// SIMATIC STEP 7 (V5.x) project 450_DMC60U
// CPU: PLC317-2DP
// station: P_ADR_BUS
// station: Hardware
// station: SINUMERIK
// station: P_ADR_BUS
// station: Hardware
// station: KSM
// station: P_ADR_BUS
// station: Hardware
// station: Rüstplatztüre
// station: P_ADR_BUS
// station: Hardware
// station: Rüstplatz_AG
// program: S7-Programm(1)
// program: S7-Programm(1)
// program: S7-Programm(1)
// program: S7-Programm(8)
// program: SINUMERIK_NX15
// program: SINAMICS_In_NCU_720

SYMBOL_TABLE
"DB_MESSAGE"	DB 2	UDT 2	// Arbeitsdaten Alarm-/Meldungserfassung
"INST_DB_TOOLING_SYSTEM"	DB 15	FB 15	// Nullpunktspannsystem
"DB_COOLANT"	DB 50	UDT 50	// Kühlmittelanlage
"INS_MESSAGE_OUT"	DB 100	FB 100	// Arbeitsdaten Alarm-/Meldungserfassung
"DB_CK_OP"	DB 101	UDT 101	// DB für Überwachung von Operanden
"DB_IN"	DB 111	DB 111	// Kommunikation - Eingänge
"DB_OUT"	DB 112	DB 112	// Kommunikation - Ausgänge
"TOOLING SYSTEM???"	FB 15	FB 15	// Nullpunktspannsystem
"MESSAGE_OUT"	FB 100	FB 100	// Ausgabe Alarm-/Betriebsmeldungen
"FLOW_CONTROL"	FC 10	FC 10	// Durchflussüberwachung
"STATUS_INDICATOR"	FC 30	FC 30
"COOLANT"	FC 50	FC 50	// Kühlmittel Druckerhöhung
"FUNCTIONS"	FC 90	FC 90	// allgemeine Funktionen
"CHANGE_BYTE"	FC 91	FC 91
"SIGNAL"	FC 92	FC 92	// allgemeine Signalverknüpfungen
"FC_CK2OP"	FC 101	FC 101	// Überwachung von 2 Operanden
"FC_CK1OP"	FC 102	FC 102	// Überwachung eines Operanden
"INPUT_MASTER"	FC 111	FC 111	// Eingänge von Mastersystem lesen
"OUTPUT_MASTER"	FC 112	FC 112	// Ausgänge an Mastersystem schreiben
"INPUT_PERIPHERIE"	FC 121	FC 121	// Eingänge von Peripherie lesen
"OUTPUT_PERIPHERIE"	FC 122	FC 122	// Ausgänge an Peripherie schreiben
"M_LOW"	M 0.0	BOOL	// Merker mit Zustand Low  "FALSE"
"M_HIGH"	M 0.1	BOOL	// Merker mit Zustand High  "TRUE"
"m_expertenbit"	M 0.2	BOOL	// Expertenbit für Fehleranzeige
"M_STARTPULSE"	M 0.5	BOOL	// Startimpuls, wird nur einmalig, für einen Zyklus gesetzt.
"m_inbetriebnahme"	M 0.6	BOOL
"m_konstruktion"	M 0.7	BOOL
"M_TAKT_0.1SEC"	M 1.0	BOOL	// Taktmerker 0.1sec/10Hz
"M_TAKT_0.2SEC"	M 1.1	BOOL	// Taktmerker 0.2sec/5Hz
"M_TAKT_0.4SEC"	M 1.2	BOOL	// Taktmerker 0.4sec/2.5Hz
"M_TAKT_0.5SEC"	M 1.3	BOOL	// Taktmerker 0.5sec/2Hz
"M_TAKT_0.8SEC"	M 1.4	BOOL	// Taktmerker 0.8sec/1.25Hz
"M_TAKT_1.0SEC"	M 1.5	BOOL	// Taktmerker 1.0sec/1Hz
"M_TAKT_1.6SEC"	M 1.6	BOOL	// Taktmerker 1.6sec/0.625Hz
"M_TAKT_2.0SEC"	M 1.7	BOOL	// Taktmerker 2.0sec/0.5Hz
"Hilfsmerker_Flanke_1"	M 10.0	BOOL
"Hilfsmerker_Flanke_2"	M 10.1	BOOL
"Hilfsmerker_Flanke_3"	M 10.3	BOOL
"Hilfsmerker_Flanke_4"	M 10.4	BOOL
"Hilfsmerker_Flanke_5"	M 10.5	BOOL
"Hilfsmerker_Flanke_6"	M 10.6	BOOL
"Hilfsmerker_KSS_aus"	M 10.7	BOOL
"Hilfsmerker_KSS_aus1"	M 11.0	BOOL
"m_sqz"	M 11.1	BOOL	// zus.Störung quittieren
"m_ilp_ventilate"	M 11.2	BOOL	// Anlage belüftet
"m_need_ventilate"	M 11.3	BOOL	// Benötigt Entlüftung
"kmsto"	M 50.0	BOOL	// Kühlmittelanlage Sammelstörung
"m_fn_m7S"	M 50.1	BOOL	// negative Flanke von M7/Spritzpistole
"m_fp_masch_on"	M 50.2	BOOL	// positive Flanke bei Maschine Ein
"m_fn_m7opendoor"	M 50.3	BOOL	// negative Flanke von M7 bei öffnen der Arbeitsraumtüre
"m50.4"	M 50.4	BOOL
"m50.5"	M 50.5	BOOL
"m50.6"	M 50.6	BOOL
"m50.7"	M 50.7	BOOL
"m51.0"	M 51.0	BOOL
"m51.1"	M 51.1	BOOL
"m51.2"	M 51.2	BOOL
"m51.3"	M 51.3	BOOL
"m51.4"	M 51.4	BOOL
"m51.5"	M 51.5	BOOL
"m51.6"	M 51.6	BOOL
"m51.7"	M 51.7	BOOL
"m52.0"	M 52.0	BOOL
"m52.1"	M 52.1	BOOL
"m52.2"	M 52.2	BOOL
"m52.3"	M 52.3	BOOL
"m52.4"	M 52.4	BOOL
"m52.5"	M 52.5	BOOL
"m52.6"	M 52.6	BOOL
"m52.7"	M 52.7	BOOL
"m53.0"	M 53.0	BOOL
"m53.1"	M 53.1	BOOL
"m53.2"	M 53.2	BOOL
"m53.3"	M 53.3	BOOL
"m53.4"	M 53.4	BOOL
"m53.5"	M 53.5	BOOL
"m53.6"	M 53.6	BOOL
"m53.7"	M 53.7	BOOL
"m54.0"	M 54.0	BOOL
"m54.1"	M 54.1	BOOL
"m54.2"	M 54.2	BOOL
"m54.3"	M 54.3	BOOL
"m54.4"	M 54.4	BOOL
"m54.5"	M 54.5	BOOL
"m54.6"	M 54.6	BOOL
"m54.7"	M 54.7	BOOL
"m55.0"	M 55.0	BOOL
"m55.1"	M 55.1	BOOL
"m55.2"	M 55.2	BOOL
"m55.3"	M 55.3	BOOL
"m55.4"	M 55.4	BOOL
"m55.5"	M 55.5	BOOL
"m55.6"	M 55.6	BOOL
"m55.7"	M 55.7	BOOL
"m56.0"	M 56.0	BOOL
"m56.1"	M 56.1	BOOL
"m56.2"	M 56.2	BOOL
"m56.3"	M 56.3	BOOL
"m56.4"	M 56.4	BOOL
"m56.5"	M 56.5	BOOL
"m56.6"	M 56.6	BOOL
"m56.7"	M 56.7	BOOL
"m57.0"	M 57.0	BOOL
"m57.1"	M 57.1	BOOL
"m57.2"	M 57.2	BOOL
"m57.3"	M 57.3	BOOL
"m57.4"	M 57.4	BOOL
"m57.5"	M 57.5	BOOL
"m57.6"	M 57.6	BOOL
"m57.7"	M 57.7	BOOL
"m_pumpe_testlauf"	M 60.0	BOOL	// Start Niederdruckpumpe (für Testlauf)
"EPX_FLOW_HD"	M 100.0	BOOL	// Durchflusswächter Kühlmittel2 (M7)
"EPX_WIREBREAK_HD"	M 100.1	BOOL	// /Durchflusswächter HD Leitungsüberwachung
"EPX_FLOW_ND"	M 100.2	BOOL	// Durchflusswächter Kühlmittel1 (M8)
"EPX_WIREBREAK_ND"	M 100.3	BOOL	// /Durchflusswächter ND Leitungsüberwachung
"EPX_ZPS_RELEASE"	M 100.4	BOOL	// Nullpunktspannsystem lösen
"EPX_ZPS_LOCK"	M 100.5	BOOL	// Nullpunktspannsystem gesperrt
"EPX_ZPS_PRESSURE_MIN1"	M 100.6	BOOL	// Nullpunktspannsystem Drucküberwachung_1 Minimaldruck (p~0) = gespannt
"EPX_ZPS_PRESSURE_MIN2"	M 100.7	BOOL	// Nullpunktspannsystem Drucküberwachung_2 Minimaldruck (p~0) = gespannt
"EPX_ZPS_PRESSURE_MAX1"	M 101.0	BOOL	// Nullpunktspannsystem Drucküberwachung_1 Maximaldruck (p=max) = gelöst
"EPX_ZPS_PRESSURE_MAX2"	M 101.1	BOOL	// Nullpunktspannsystem Drucküberwachung_2 Maximaldruck (p=max) = gelöst
"EPX_COOLANT_LIMIT_VALUE"	M 101.2	BOOL	// /Füllstandsüberwachung im Sammelbehälter
"EPX_LUBRICATION_LEVEL"	M 101.3	BOOL	// Füllstandsüberwachung Schmierstoffaggregat
"EPX_ZPS_MODE_AUTO"	M 101.4	BOOL	// Nullpunktspannsystem in Betriebsart Automatik = Ansteuerung durch ext. Einheit
"EPX_ZPS_INTERLOCK_MIN1"	M 101.5	BOOL	// Nullpunktspannsystem - Verriegelungskontrolle Druck ~0 (drucklos)
"EPX_ZPS_INTERLOCK_MAX1"	M 101.6	BOOL	// Nullpunktspannsystem - Verriegelungskontrolle Druck vorhanden (=verriegelt)
"EPX_ZPS_DISTANCE_P_MIN1"	M 101.7	BOOL	// Nullpunktspannsystem - Auflagenkontrolle Druck ~0 (drucklos)
"EPX_ZPS_DISTANCE_P_MAX1"	M 102.0	BOOL	// Nullpunktspannsystem - Auflagenkontrolle Druck erreicht (Präzision vorhanden)
"EPX_ALARM_QUIT"	M 102.1	BOOL	// Rücksetzen der Fehlermeldung (z.B. Akustik)
"EPX_EL-CABINETDOOR1_OPEN"	M 102.2	BOOL	// Schaltschranktür(-kombination)_1 der Werkzeugmaschine geöffnet
"EPX_EL-CABINETDOOR2_OPEN"	M 102.3	BOOL	// Schaltschranktür(-kombination)_2 der Werkzeugmaschine geöffnet
"EPX_EL-CABINETDOOR5_OPEN"	M 102.4	BOOL	// Schaltschranktür(-kombination)_1 der Kühlschmierstoffanlage geöffnet
"EPX_EL_CABINET_TEMP_1"	M 102.5	BOOL	// Uebertemperatur Schaltschrank Werkzeugmaschine
"EPX_EL_CABINET_TEMP_2"	M 102.6	BOOL	// Grenzwertmeldung Schaltschranktemperatur Werkzeugmaschine
"EPX_EL-CABINETDOOR3_OPEN"	M 102.7	BOOL	// Schaltschranktür(-kombination)_3 der Werkzeugmaschine geöffnet
"EPX_SO_APC_POS_180"	M 103.0	BOOL	// Palettenwechsler Stellung 180 Grad (Palette_2 im Arbeitsraum)
"EPX_SO_APC_POS_0"	M 103.1	BOOL	// Palettenwechsler Stellung 0 Grad (Palette_1 im Arbeitsraum)
"EPX_VCS_MODE_MIXED"	M 103.2	BOOL	// Anwahl Betriebsart <Vakuumsystem Mischbetrieb> aktiv
"EPX_VCS_MODE_VACUUM"	M 103.3	BOOL	// Anwahl Betriebsart <Vakuumsystem Vollwechsel> aktiv
"EPX_VCS_MODE_OFF"	M 103.4	BOOL	// Anwahl Betriebsart <Vakuumsystem Aus>
"EPX_VCS_READY_1"	M 103.5	BOOL	// Betriebsbereitmeldung Vakuumsystem (Arbeitsraum) z.B. Leistungssschalter, ...
"EPX_VCS_READY_2"	M 103.6	BOOL	// Betriebsbereitmeldung Vakuumsystem (Rüstplatz) z.B. Leistungssschalter, ...
"EPX_VCS_RELEASE_FIXTURE2"	M 103.7	BOOL	// Vakuumspannsystem am Rüstplatz lösen
"EPX_VCS_FIXTURE1_1_P=0"	M 104.0	BOOL	// Vakuumspannsystem im Arbeitsraum Drucklos (=gelöst)
"EPX_VCS_FIXTURE1_2_P=0"	M 104.1	BOOL	// Vakuumspannsystem im Arbeitsraum Drucklos (=gelöst)
"EPX_VCS_FIXTURE2_1_P=0"	M 104.2	BOOL	// Vakuumspannsystem am Rüstplatz Drucklos (=gelöst)
"EPX_VCS_FIXTURE1_1_P=MAX"	M 104.3	BOOL	// Vakuumspannsystem im Arbeitsraum gespannt (eingestellter Sollwert erreicht)
"EPX_VCS_FIXTURE2_1_P=MAX"	M 104.4	BOOL	// Vakuumspannsystem am Rüstplatz gespannt (eingestellter Sollwert erreicht)
"EPX_NEG_HYD_FILTERALARM1"	M 104.5	BOOL	// Filterverschmutzung Hydraulikfilter-Maschine (Alarm 100%)
"EPX_NEG_HYD_FILTERWARN1"	M 104.6	BOOL	// Filterverschmutzung Hydraulikfilter-Maschine (Warnung 75%)
"EPX_NEG_FUSE_AIRFILTER"	M 104.7	BOOL	// Auswertung Leistungsschalter des Nebelabscheiders/Absaugung
"EPX_POWER_AIRFILTER"	M 105.0	BOOL	// Überwachung Ansteuerung Nebelabscheider
"EPX_MACHINE_ON_K1"	M 105.1	BOOL	// "Maschine Ein"-Signal an Kühlschmierstoffanlage (kein Not-Aus)
"EPX_WORKROOM_CLOSED_K1"	M 105.2	BOOL	// "Arbeitsraumtüren geschlossen"-Signal an Kühlschmierstoffanlage
"EPX_NEG_COO_MESSAGE"	M 105.3	BOOL	// Warnmeldung von Kühlschmierstoffanlage
"EPX_NEG_COO_ALARM"	M 105.4	BOOL	// Störung, Alarm von Kühlschmierstoffanlage
"EPX_COO_ACK_COOLANT2.2"	M 105.5	BOOL	// Rückmeldung wenn Druckstufe_2 von Kühlmittel_2 erreicht wurde (YD-Anlauf)
"EPX_COO_MAINVALVE_CLOSED"	M 105.6	BOOL	// Kühlschmierstoffzufuhr Haupt-/Zentralventil geschlossen
"EPX_COO_PRESSURE_P=MAX"	M 105.7	BOOL	// Kühlschmierstoffzufuhr Drucküberwachung
"EPX_COO_MAIN_FLOW"	M 106.0	BOOL	// Kühlschmierstoffzufuhr Durchflussüberwachung
"EPX_COO_LIMITVALUE_K5"	M 106.1	BOOL	// Grenzwertmeldung aus Sammelbehälter (SPF) z.B. von WHG-Sonde
"EPX_NEG_COO_FILTALARM2.2"	M 106.2	BOOL	// Filterverschmutzung Feinfilter Alarmmeldung für KSS-Zufuhr_2 (IKZ)-Druckstufe_2
"EPX_COO_FILTWARN2.2"	M 106.3	BOOL	// Filterverschmutzung Feinfilter Warnmeldung für KSS-Zufuhr_2 (IKZ) - Druckstufe_2
"EPX_VCS_RELEASE_FIXTURE1"	M 106.4	BOOL	// Vakuumspannsystem im Arbeitsraum lösen
"m106.5"	M 106.5	BOOL
"m106.6"	M 106.6	BOOL
"m106.7"	M 106.7	BOOL
"APX_SIGNAL_TOWER_GN"	M 180.0	BOOL	// Signalleuchte (Ampel) Element: GRÜN (GN)
"APX_SIGNAL_TOWER_YE"	M 180.1	BOOL	// Signalleuchte (Ampel) Element: GELB (YE)
"APX_SIGNAL_TOWER_RD"	M 180.2	BOOL	// Signalleuchte (Ampel) Element: ROT (RD)
"APX_BDE_AXIS_SPINDLE"	M 180.3	BOOL	// mindestens 1Achse und Spindel aktiv
"APX_BDE_MACHINE_ON"	M 180.4	BOOL	// Maschine Ein (kein Not-Aus)
"APX_MODE_MANUAL"	M 180.5	BOOL	// Betriebsart "MANUAL"
"APX_MODE_TEACH_IN"	M 180.6	BOOL	// Betriebsart "TEACH IN"
"APX_MODE_AUTOMATIK"	M 180.7	BOOL	// Betriebsart "AUTOMATIK"
"APX_FEEDRATE>X%"	M 181.0	BOOL	// Vorschubpotentiometer größer Wert "X"
"APX_CNC_ERROR"	M 181.1	BOOL	// Fehlermeldung CNC
"APX_PROG_STOP"	M 181.2	BOOL	// Programm Halt
"APX_PROG_RUN"	M 181.3	BOOL	// Programm läuft
"APX_CNC_READY2RUN"	M 181.4	BOOL	// CNC-Betriebsbereit
"APX_ZPS_BLOW_OUT"	M 181.5	BOOL	// Nullpunktspannsystem Blasluft (Reinigung)
"APX_ZPS_STATUS"	M 181.6	BOOL	// Nullpunktspannsystem Statusmeldung Betriebsartenanzeige
"APX_ZPS_RELEASE1"	M 181.7	BOOL	// Nullpunktspannsystem lösen (Ventil_1)
"APX_ZPS_RELEASE2"	M 182.0	BOOL	// Nullpunktspannsystem lösen (Ventil_2)
"APX_ZPS_INTERLOCK1"	M 182.4	BOOL	// Nullpunktspannsystem - Ansteuerung (Ventil) für Verriegelungskontrolle
"APX_ZPS_DISTANCE_CHECK1"	M 182.5	BOOL	// Nullpunktspannsystem - Ansteuerung (Ventil) für Auflagenkontrolle
"APX_WORKPIECE_COUNT"	M 182.6	BOOL	// Werkstück Zählimpuls
"APX_PRODUCTION"	M 182.7	BOOL	// Produktionssignal der Werkzeugmaschine/Maschine Produziert (Programm läuft)
"APX_PALLET-NR_BIT0"	M 183.0	BOOL	// Nummer der Palette Arbeitsraum 2^0 (=1)
"APX_PALLET-NR_BIT1"	M 183.1	BOOL	// Nummer der Palette Arbeitsraum 2^1 (=2)
"APX_PALLET-NR_BIT2"	M 183.2	BOOL	// Nummer der Palette Arbeitsraum 2^2 (=4)
"APX_PALLET-NR_BIT3"	M 183.3	BOOL	// Nummer der Palette Arbeitsraum 2^3 (=8)
"APX_ALARM_LIGHT"	M 183.4	BOOL	// Optische Anzeige einer Fehlermeldung
"APX_AUDIBLE_ALARM"	M 183.5	BOOL	// Akustische Ausgabe einer Fehlermeldung
"APX_VCS_RELEASE_FIXTURE1"	M 183.6	BOOL	// Vakuumspannsystem im Arbeitsraum Lösen (=drucklos)
"APX_VCS_RELEASE_FIXTURE2"	M 183.7	BOOL	// Vakuumspannsystem am Rüstplatz Lösen (=drucklos)
"APX_AIRFILTER_ON"	M 184.0	BOOL	// Aktivieren und evtl.verzögertes Abschalten des Nebelabscheiders
"APX_COO_COOLANT1_(M8)"	M 184.1	BOOL	// Aktivierung Kühlschmierstoffzufuhr_1 (externe - Spritzdüsen)
"APX_COO_PALLET_CARRIER"	M 184.2	BOOL	// Aktivierung Spänespülung Palettenträger (Umschaltung IKZ)
"APX_COO_WORKPIECE_1"	M 184.3	BOOL	// Aktivierung Spänespülung Werkstückreinigung (Dachspülung)
"APX_COO_SPRAYGUN"	M 184.4	BOOL	// Aktivierung Spritzpistole, Spülpistole
"APX_COO_WORKROOMDOOR"	M 184.5	BOOL	// Aktivierung Spänespülung Kabinentüre, Arbeitsraumtüre
"APX_COO_COOLANT2.2"	M 184.6	BOOL	// Aktivierung Kühlschmierstoffzufuhr_2 (IKZ) - Druckstufe_2
"APX_COO_MAINVALVE"	M 184.7	BOOL	// Aktivierung Kühlschmierstoffzufuhr Haupt-/Zentralventil
"APX_COO_LOCKVALVE_RET"	M 185.0	BOOL	// Aktivierung Sperrventil für Kühlschmierstoffrückführung aus Sammelbehälter (SPF)
"APX_ALARM_RESET"	M 185.1	BOOL	// Bei Betätigung der "Alarm-Quit-Taste (F10)" wird Ausgang gesetzt
"APX_NO_MACHINING"	M 185.2	BOOL	// MDE/BDE: keine Bearbeitung
"APX_INTO_PRODUCTION"	M 185.3	BOOL	// MDE/BDE: Produktionssignal
"APX_PROG_END"	M 185.4	BOOL	// Programm Ende
"m185.5"	M 185.5	BOOL
"m185.6"	M 185.6	BOOL
"m185.7"	M 185.7	BOOL
"APX_COO_LOCKVALVE2.2"	M 188.0	BOOL	// Aktivierung Sperrventil für Kühlschmierstoffzufuhr - Druckstufe_2
"QpxFlushSetUpStation"	M 197.0	BOOL	// Spänespülung am Rüstplatz (Spannvorrichtung, Werkstück, ...)
"m_AkTime"	MD 12	TIME	// ausgeleseneSysZeitVonTime_tck SFC64
"APW_COO_PRESS_VALUE2.2"	MW 186	WORD	// Sollwertvorgabe für Druckvorwahl Kühlmittel_2 (inner Kühlschmierstoffzufuhr)
"CYCL_EXC"	OB 1	OB 1	// Cycle Execution
"I/O_FLT1"	OB 82	OB 82	// I/O Point Fault 1
"CPU_FLT"	OB 84	OB 84	// CPU Fault
"OBNL_FLT"	OB 85	OB 85	// OB Not Loaded Fault
"RACK_FLT"	OB 86	OB 86	// Loss of Rack Fault
"START"	OB 100	OB 100	// Anlauf OB
"PROG_ERR"	OB 121	OB 121	// Programming Error
"MOD_ERR"	OB 122	OB 122	// Module Access Error
"BLKMOV"	SFC 20	SFC 20	// Copy Variables
"TIME_TCK"	SFC 64	SFC 64	// Time tics of period 10 ms
"t0"	T 0	TIMER	// 840D Grundprg.
"t1"	T 1	TIMER	// 840D Grundprg.
"t2"	T 2	TIMER	// 840D Grundprg.
"t3"	T 3	TIMER	// 840D Grundprg.
"t4"	T 4	TIMER	// 840D Grundprg.
"t5"	T 5	TIMER	// 840D Grundprg.
"t6"	T 6	TIMER	// 840D Grundprg.
"t7"	T 7	TIMER	// 840D Grundprg.
"t8"	T 8	TIMER	// 840D Grundprg.
"t9"	T 9	TIMER	// 840D Grundprg.
"t10"	T 10	TIMER
"Hilfs_Timer_1"	T 11	TIMER
"Hilfs_Timer_2"	T 12	TIMER
"Hilfs_Timer_3"	T 13	TIMER
"Hilfs_Timer_4"	T 14	TIMER
"Hilfs_Timer_5"	T 15	TIMER
"Hilfs_Timer_6"	T 16	TIMER
"t_sp_twa"	T 17	TIMER	// se Nullspannsystem Schrittkette Wartezeit
"t_sp_tue"	T 18	TIMER	// se Nullspannsystem Schrittkette Überwachungszeit (Reserve)
"t_nspgs"	T 19	TIMER	// se Nullspannsystem gespannt
"t_nspgsa"	T 20	TIMER	// sa Nullspannsystem gespannt
"t_nspgl"	T 21	TIMER	// se Nullspannsystem gelöst
"t_nspgla"	T 22	TIMER	// sa Nullspannsystem gelöst
"t23"	T 23	TIMER
"t24"	T 24	TIMER
"t_toggle"	T 25	TIMER	// Zeit für FB100 Anzeigeintervall
"t26"	T 26	TIMER
"t27"	T 27	TIMER
"t28"	T 28	TIMER
"t29"	T 29	TIMER
"t30"	T 30	TIMER
"t31"	T 31	TIMER
"ta_pressureless"	T 32	TIMER	// Belüften der Druckerhöhungsstation nach M7
"t33"	T 33	TIMER
"t34"	T 34	TIMER
"t35"	T 35	TIMER
"t36"	T 36	TIMER
"t37"	T 37	TIMER
"t38"	T 38	TIMER
"t39"	T 39	TIMER
"t40"	T 40	TIMER
"t41"	T 41	TIMER
"t42"	T 42	TIMER
"t43"	T 43	TIMER
"t44"	T 44	TIMER
"t45"	T 45	TIMER
"t46"	T 46	TIMER
"t47"	T 47	TIMER
"t48"	T 48	TIMER
"t49"	T 49	TIMER
"ta_kss_mainvalve"	T 50	TIMER	// Ausschaltverzögerung Km-Hauptventil ein
"t_kmfue"	T 51	TIMER	// se Überwachung Kühlmittelfilter
"t_kmFSp"	T 52	TIMER	// sa Km-Hochdruck-Sperrventil ein (=Frg.Hochdruck)
"t_kmrv"	T 53	TIMER	// se KmRückförderventil=Sperrventil öffnen
"ta_kss_km1"	T 54	TIMER	// Ausschaltverzögerung Kühlmittelanwahl (AKZ = M8)
"ta_kss_spraygun"	T 55	TIMER	// Ausschaltverzögerung für Spritzpistole
"ta_kss_workroomdoor"	T 56	TIMER	// Ausschaltverzögerung für Türspülung
"ta_kss_workpiece1"	T 57	TIMER	// Ausschaltverzögerung für Dachspülung (Werkstückspülung)
"te_aktiv_monit_pressure"	T 58	TIMER	// Einschaltverzögerung für Aktivierung Drucküberwachung
"ta_kss_setupstation"	T 59	TIMER	// Ausschaltverzögerung für Rüstplatzspülung(Vorrichtung)
"UDT_MESSAGE"	UDT 2	UDT 2	// UDT zu DB2 (Datenformat für Meldungen)
"UDT_COOLANT"	UDT 50	UDT 50	// UDT zu DB_COOLANT
"UDT101"	UDT 101	UDT 101
"UDT1010"	UDT 1010	UDT 1010	// UDT für UDT 101
"VAT_IN_dbw0"	VAT 1	
"VAT_IN_dbw2"	VAT 2	
"VAT_IN_dbw4"	VAT 3	
"VAT_IN_dbw6"	VAT 4	
"VAT_IN_dbw10_12"	VAT 5	
"VAT_OUT_dbw2"	VAT 6	
"VAT_OUT_dbw0"	VAT 7	
"VAT_PER"	VAT 8	
"VAT_MESSAGE"	VAT 9		// Meldungen, Alarme
"V_Nps0"	VAT 10		// Nullspannsystem
"V_allg"	VAT 11	
"VATksaÜW"	VAT 12	
"VAT_OUT_dbw6"	VAT 13	
END_SYMBOL_TABLE

TYPE "UDT_MESSAGE"	// UDT 2
AUTHOR : SPAC_slh
VERSION : 0.0
  STRUCT
   ALARM_001 : BOOL ;	//Schaltschranktemperatur zu hoch
   ALARM_002 : BOOL ;	//Schaltschranktemperatur - Grenzwert überschritten
   F003 : BOOL ;	//1-
   F004 : BOOL ;	//1-
   F005 : BOOL ;	//1-
   F006 : BOOL ;	//1-
   F007 : BOOL ;	//1-
   F008 : BOOL ;	//1-
   F009 : BOOL ;	//1-
   F010 : BOOL ;	//1-
   F011 : BOOL ;	//1-
   F012 : BOOL ;	//1-
   F013 : BOOL ;	//1-
   F014 : BOOL ;	//1-
   F015 : BOOL ;	//1-
   F016 : BOOL ;	//1-
   F017 : BOOL ;	//Nullpunktspannsysten Laufzeitfehler lösen_1
   F018 : BOOL ;	//Spanner 1 LzFehler spannen
   F019 : BOOL ;	//Spanner 1 Fehler Endlage gelöst
   F020 : BOOL ;	//Spanner 1 Fehler Endlage gespannt
   F021 : BOOL ;	//Spanner 1 Fehler Paarüberwachung
   F022 : BOOL ;	//Nullpunktspannsysten Laufzeitfehler lösen_2
   F023 : BOOL ;	//Spanner 2 LzFehler spannen
   F024 : BOOL ;	//Spanner 2 Fehler Endlage gelöst
   F025 : BOOL ;	//Spanner 2 Fehler Endlage gespannt
   F026 : BOOL ;	//Spanner 2 Fehler Paarüberwachung
   F027 : BOOL ;	//Auflagektrl.LzFehler bei einschalten
   F028 : BOOL ;	//Auflagektrl.LzFehler bei ausschalten
   F029 : BOOL ;	//Auflagektrl.Fehler Endlage Druck erreicht
   F030 : BOOL ;	//Auflagektrl.Fehler Endlage Drucklos
   F031 : BOOL ;	//Auflagektrl.Fehler Paarüberwachung
   F032 : BOOL ;	//Verriegelungsktrl.LzFehler bei einschalten
   F033 : BOOL ;	//Verriegelungsktrl.LzFehler bei ausschalten
   F034 : BOOL ;	//Verriegelungsktrl.Fehler Endlage Druck erreicht
   F035 : BOOL ;	//Verriegelungsktrl.Fehler Endlage Drucklos
   F036 : BOOL ;	//Verriegelungsktrl.Fehler Paarüberwachung
   F037 : BOOL ;	//1-
   F038 : BOOL ;	//1-
   F039 : BOOL ;	//1-
   F040 : BOOL ;	//1-
   F041 : BOOL ;	//1-
   F042 : BOOL ;	//1-
   F043 : BOOL ;	//1-
   F044 : BOOL ;	//1-
   F045 : BOOL ;	//1-
   F046 : BOOL ;	//1-
   F047 : BOOL ;	//1-
   F048 : BOOL ;	//1-
   F049 : BOOL ;	//1-
   F050 : BOOL ;	//1-
   F051 : BOOL ;	//1-
   F052 : BOOL ;	//1-
   F053 : BOOL ;	//1-
   F054 : BOOL ;	//1-
   F055 : BOOL ;	//1-
   F056 : BOOL ;	//1-
   F057 : BOOL ;	//1-
   F058 : BOOL ;	//1-
   F059 : BOOL ;	//1-
   F060 : BOOL ;	//1-
   F061 : BOOL ;	//1-
   F062 : BOOL ;	//1-
   F063 : BOOL ;	//1-
   F064 : BOOL ;	//1-
   F065 : BOOL ;	//1-
   F066 : BOOL ;	//1-
   F067 : BOOL ;	//1-
   F068 : BOOL ;	//1-
   F069 : BOOL ;	//1-
   F070 : BOOL ;	//1-
   F071 : BOOL ;	//1-
   F072 : BOOL ;	//1-
   F073 : BOOL ;	//1-
   F074 : BOOL ;	//1-
   F075 : BOOL ;	//1-
   F076 : BOOL ;	//1-
   F077 : BOOL ;	//1-
   F078 : BOOL ;	//1-
   F079 : BOOL ;	//1-
   F080 : BOOL ;	//1-
   F081 : BOOL ;	//1-
   F082 : BOOL ;	//1-
   F083 : BOOL ;	//1-
   F084 : BOOL ;	//1-
   F085 : BOOL ;	//1-
   F086 : BOOL ;	//1-
   F087 : BOOL ;	//1-
   F088 : BOOL ;	//1-
   F089 : BOOL ;	//1-
   F090 : BOOL ;	//1-
   F091 : BOOL ;	//1-
   F092 : BOOL ;	//1-
   F093 : BOOL ;	//1-
   F094 : BOOL ;	//1-
   F095 : BOOL ;	//1-
   F096 : BOOL ;	//1-
   F097 : BOOL ;	//Km-Hautpventil nicht offen, Eingang meldet "zu", muss 0-Signal melden
   F098 : BOOL ;	//Km-Hautpventil schließt nicht, Eingang muss 1-Signal melden
   F099 : BOOL ;	//WHG-Alarm
   F100 : BOOL ;	//Reserve Km-Alarm
   F101 : BOOL ;	//Km-Systemdruck fehlt, Eingang muss 1-Signal melden
   F102 : BOOL ;	//Km-Systemdruck, Druckschalter defekt, Eingang muss 0-Signal melden
   F103 : BOOL ;	//Km-Durchfluss fehlt, Eingang muss 1-Signal melden
   F104 : BOOL ;	//Km-Durchfluss-Schalter defekt, Eingang muss 0-Signal melden
   F105 : BOOL ;	//Kühlmittelfeinfilter verschmutzt
   F106 : BOOL ;	//Kühlmittelfeinfilter Schalterpaarüberwachung
   F107 : BOOL ;	//Reserve Km-Alarm
   F108 : BOOL ;	//Reserve Km-Alarm
   F109 : BOOL ;	//Reserve Km-Alarm
   F110 : BOOL ;	//Reserve Km-Alarm
   F111 : BOOL ;	//Reserve Km-Alarm
   F112 : BOOL ;	//Reserve Km-Alarm
   F113 : BOOL ;	//1-
   F114 : BOOL ;	//1-
   F115 : BOOL ;	//1-
   F116 : BOOL ;	//1-
   F117 : BOOL ;	//1-
   F118 : BOOL ;	//1-
   F119 : BOOL ;	//1-
   F120 : BOOL ;	//1-
   F121 : BOOL ;	//1-
   F122 : BOOL ;	//1-
   F123 : BOOL ;	//1-
   F124 : BOOL ;	//1-
   F125 : BOOL ;	//1-
   F126 : BOOL ;	//1-
   F127 : BOOL ;	//1-
   F128 : BOOL ;	//1-
   F129 : BOOL ;	//1-
   F130 : BOOL ;	//1-
   F131 : BOOL ;	//1-
   F132 : BOOL ;	//1-
   F133 : BOOL ;	//1-
   F134 : BOOL ;	//1-
   F135 : BOOL ;	//1-
   F136 : BOOL ;	//1-
   F137 : BOOL ;	//1-
   F138 : BOOL ;	//1-
   F139 : BOOL ;	//1-
   F140 : BOOL ;	//1-
   F141 : BOOL ;	//1-
   F142 : BOOL ;	//1-
   F143 : BOOL ;	//1-
   F144 : BOOL ;	//1-
   F145 : BOOL ;	//1-
   F146 : BOOL ;	//1-
   F147 : BOOL ;	//1-
   F148 : BOOL ;	//1-
   F149 : BOOL ;	//1-
   F150 : BOOL ;	//1-
   F151 : BOOL ;	//1-
   F152 : BOOL ;	//1-
   F153 : BOOL ;	//1-
   F154 : BOOL ;	//1-
   F155 : BOOL ;	//1-
   F156 : BOOL ;	//1-
   F157 : BOOL ;	//1-
   F158 : BOOL ;	//1-
   F159 : BOOL ;	//1-
   F160 : BOOL ;	//1-
   F161 : BOOL ;	//1-
   F162 : BOOL ;	//1-
   F163 : BOOL ;	//1-
   F164 : BOOL ;	//1-
   F165 : BOOL ;	//1-
   F166 : BOOL ;	//1-
   F167 : BOOL ;	//1-
   F168 : BOOL ;	//1-
   F169 : BOOL ;	//1-
   F170 : BOOL ;	//1-
   F171 : BOOL ;	//1-
   F172 : BOOL ;	//1-
   F173 : BOOL ;	//1-
   F174 : BOOL ;	//1-
   F175 : BOOL ;	//1-
   F176 : BOOL ;	//1-
   F177 : BOOL ;	//1-
   F178 : BOOL ;	//1-
   F179 : BOOL ;	//1-
   F180 : BOOL ;	//1-
   F181 : BOOL ;	//1-
   F182 : BOOL ;	//1-
   F183 : BOOL ;	//1-
   F184 : BOOL ;	//1-
   F185 : BOOL ;	//1-
   F186 : BOOL ;	//1-
   F187 : BOOL ;	//1-
   F188 : BOOL ;	//1-
   F189 : BOOL ;	//1-
   F190 : BOOL ;	//1-
   F191 : BOOL ;	//1-
   F192 : BOOL ;	//1-
   F193 : BOOL ;	//1-
   F194 : BOOL ;	//1-
   F195 : BOOL ;	//1-
   F196 : BOOL ;	//1-
   F197 : BOOL ;	//1-
   F198 : BOOL ;	//1-
   F199 : BOOL ;	//1-
   F200 : BOOL ;	//1-
   F201 : BOOL ;	//1-
   F202 : BOOL ;	//1-
   F203 : BOOL ;	//1-
   F204 : BOOL ;	//1-
   F205 : BOOL ;	//1-
   F206 : BOOL ;	//1-
   F207 : BOOL ;	//1-
   F208 : BOOL ;	//1-
   F209 : BOOL ;	//1-
   F210 : BOOL ;	//1-
   F211 : BOOL ;	//1-
   F212 : BOOL ;	//1-
   F213 : BOOL ;	//1-
   F214 : BOOL ;	//1-
   F215 : BOOL ;	//1-
   F216 : BOOL ;	//1-
   F217 : BOOL ;	//1-
   F218 : BOOL ;	//1-
   F219 : BOOL ;	//1-
   F220 : BOOL ;	//1-
   F221 : BOOL ;	//1-
   F222 : BOOL ;	//1-
   F223 : BOOL ;	//1-
   F224 : BOOL ;	//1-
   F225 : BOOL ;	//1-
   F226 : BOOL ;	//1-
   F227 : BOOL ;	//1-
   F228 : BOOL ;	//1-
   F229 : BOOL ;	//1-
   F230 : BOOL ;	//1-
   F231 : BOOL ;	//1-
   F232 : BOOL ;	//1-
   F233 : BOOL ;	//1-
   F234 : BOOL ;	//1-
   F235 : BOOL ;	//1-
   F236 : BOOL ;	//1-
   F237 : BOOL ;	//1-
   F238 : BOOL ;	//1-
   F239 : BOOL ;	//1-
   F240 : BOOL ;	//1-
   F241 : BOOL ;	//1-
   F242 : BOOL ;	//1-
   F243 : BOOL ;	//1-
   F244 : BOOL ;	//1-
   F245 : BOOL ;	//1-
   F246 : BOOL ;	//1-
   F247 : BOOL ;	//1-
   F248 : BOOL ;	//1-
   F249 : BOOL ;	//1-
   F250 : BOOL ;	//1-
   F251 : BOOL ;	//1-
   F252 : BOOL ;	//1-
   F253 : BOOL ;	//1-
   F254 : BOOL ;	//1-
   F255 : BOOL ;	//1-
   F256 : BOOL ;	//1-
   F257 : BOOL ;	//1-
   F258 : BOOL ;	//1-
   F259 : BOOL ;	//1-
   F260 : BOOL ;	//1-
   F261 : BOOL ;	//1-
   F262 : BOOL ;	//1-
   F263 : BOOL ;	//1-
   F264 : BOOL ;	//1-
   F265 : BOOL ;	//1-
   F266 : BOOL ;	//1-
   F267 : BOOL ;	//1-
   F268 : BOOL ;	//1-
   F269 : BOOL ;	//1-
   F270 : BOOL ;	//1-
   F271 : BOOL ;	//1-
   F272 : BOOL ;	//1-
   F273 : BOOL ;	//1-
   F274 : BOOL ;	//1-
   F275 : BOOL ;	//1-
   F276 : BOOL ;	//1-
   F277 : BOOL ;	//1-
   F278 : BOOL ;	//1-
   F279 : BOOL ;	//1-
   F280 : BOOL ;	//1-
   F281 : BOOL ;	//1-
   F282 : BOOL ;	//1-
   F283 : BOOL ;	//1-
   F284 : BOOL ;	//1-
   F285 : BOOL ;	//1-
   F286 : BOOL ;	//1-
   F287 : BOOL ;	//1-
   F288 : BOOL ;	//1-
   F289 : BOOL ;	//1-
   F290 : BOOL ;	//1-
   F291 : BOOL ;	//1-
   F292 : BOOL ;	//1-
   F293 : BOOL ;	//1-
   F294 : BOOL ;	//1-
   F295 : BOOL ;	//1-
   F296 : BOOL ;	//1-
   F297 : BOOL ;	//1-
   F298 : BOOL ;	//1-
   F299 : BOOL ;	//1-
   F300 : BOOL ;	//1-
   F301 : BOOL ;	//1-
   F302 : BOOL ;	//1-
   F303 : BOOL ;	//1-
   F304 : BOOL ;	//1-
   F305 : BOOL ;	//1-
   F306 : BOOL ;	//1-
   F307 : BOOL ;	//1-
   F308 : BOOL ;	//1-
   F309 : BOOL ;	//1-
   F310 : BOOL ;	//1-
   F311 : BOOL ;	//1-
   F312 : BOOL ;	//1-
   F313 : BOOL ;	//1-
   F314 : BOOL ;	//1-
   F315 : BOOL ;	//1-
   F316 : BOOL ;	//1-
   F317 : BOOL ;	//1-
   F318 : BOOL ;	//1-
   F319 : BOOL ;	//1-
   F320 : BOOL ;	//1-
   F321 : BOOL ;	//1-
   F322 : BOOL ;	//1-
   F323 : BOOL ;	//1-
   F324 : BOOL ;	//1-
   F325 : BOOL ;	//1-
   F326 : BOOL ;	//1-
   F327 : BOOL ;	//1-
   F328 : BOOL ;	//1-
   F329 : BOOL ;	//1-
   F330 : BOOL ;	//1-
   F331 : BOOL ;	//1-
   F332 : BOOL ;	//1-
   F333 : BOOL ;	//1-
   F334 : BOOL ;	//1-
   F335 : BOOL ;	//1-
   F336 : BOOL ;	//1-
   F337 : BOOL ;	//1-
   F338 : BOOL ;	//1-
   F339 : BOOL ;	//1-
   F340 : BOOL ;	//1-
   F341 : BOOL ;	//1-
   F342 : BOOL ;	//1-
   F343 : BOOL ;	//1-
   F344 : BOOL ;	//1-
   F345 : BOOL ;	//1-
   F346 : BOOL ;	//1-
   F347 : BOOL ;	//1-
   F348 : BOOL ;	//1-
   F349 : BOOL ;	//1-
   F350 : BOOL ;	//1-
   F351 : BOOL ;	//1-
   F352 : BOOL ;	//1-
   F353 : BOOL ;	//1-
   F354 : BOOL ;	//1-
   F355 : BOOL ;	//1-
   F356 : BOOL ;	//1-
   F357 : BOOL ;	//1-
   F358 : BOOL ;	//1-
   F359 : BOOL ;	//1-
   F360 : BOOL ;	//1-
   F361 : BOOL ;	//1-
   F362 : BOOL ;	//1-
   F363 : BOOL ;	//1-
   F364 : BOOL ;	//1-
   F365 : BOOL ;	//1-
   F366 : BOOL ;	//1-
   F367 : BOOL ;	//1-
   F368 : BOOL ;	//1-
   F369 : BOOL ;	//1-
   F370 : BOOL ;	//1-
   F371 : BOOL ;	//1-
   F372 : BOOL ;	//1-
   F373 : BOOL ;	//1-
   F374 : BOOL ;	//1-
   F375 : BOOL ;	//1-
   F376 : BOOL ;	//1-
   F377 : BOOL ;	//1-
   F378 : BOOL ;	//1-
   F379 : BOOL ;	//1-
   F380 : BOOL ;	//1-
   F381 : BOOL ;	//1-
   F382 : BOOL ;	//1-
   F383 : BOOL ;	//1-
   F384 : BOOL ;	//1-
   F385 : BOOL ;	//1-
   F386 : BOOL ;	//1-
   F387 : BOOL ;	//1-
   F388 : BOOL ;	//1-
   F389 : BOOL ;	//1-
   F390 : BOOL ;	//1-
   F391 : BOOL ;	//1-
   F392 : BOOL ;	//1-
   F393 : BOOL ;	//1-
   F394 : BOOL ;	//1-
   F395 : BOOL ;	//1-
   F396 : BOOL ;	//1-
   F397 : BOOL ;	//1-
   F398 : BOOL ;	//1-
   F399 : BOOL ;	//1-
   F400 : BOOL ;	//1-
   F401 : BOOL ;	//1-
   F402 : BOOL ;	//1-
   F403 : BOOL ;	//1-
   F404 : BOOL ;	//1-
   F405 : BOOL ;	//1-
   F406 : BOOL ;	//1-
   F407 : BOOL ;	//1-
   F408 : BOOL ;	//1-
   F409 : BOOL ;	//1-
   F410 : BOOL ;	//1-
   F411 : BOOL ;	//1-
   F412 : BOOL ;	//1-
   F413 : BOOL ;	//1-
   F414 : BOOL ;	//1-
   F415 : BOOL ;	//1-
   F416 : BOOL ;	//1-
   F417 : BOOL ;	//1-
   F418 : BOOL ;	//1-
   F419 : BOOL ;	//1-
   F420 : BOOL ;	//1-
   F421 : BOOL ;	//1-
   F422 : BOOL ;	//1-
   F423 : BOOL ;	//1-
   F424 : BOOL ;	//1-
   F425 : BOOL ;	//1-
   F426 : BOOL ;	//1-
   F427 : BOOL ;	//1-
   F428 : BOOL ;	//1-
   F429 : BOOL ;	//1-
   F430 : BOOL ;	//1-
   F431 : BOOL ;	//1-
   F432 : BOOL ;	//1-
   F433 : BOOL ;	//1-
   F434 : BOOL ;	//1-
   F435 : BOOL ;	//1-
   F436 : BOOL ;	//1-
   F437 : BOOL ;	//1-
   F438 : BOOL ;	//1-
   F439 : BOOL ;	//1-
   F440 : BOOL ;	//1-
   F441 : BOOL ;	//1-
   F442 : BOOL ;	//1-
   F443 : BOOL ;	//1-
   F444 : BOOL ;	//1-
   F445 : BOOL ;	//1-
   F446 : BOOL ;	//1-
   F447 : BOOL ;	//1-
   F448 : BOOL ;	//1-
   F449 : BOOL ;	//1-
   F450 : BOOL ;	//1-
   F451 : BOOL ;	//1-
   F452 : BOOL ;	//1-
   F453 : BOOL ;	//1-
   F454 : BOOL ;	//1-
   F455 : BOOL ;	//1-
   F456 : BOOL ;	//1-
   F457 : BOOL ;	//1-
   F458 : BOOL ;	//1-
   F459 : BOOL ;	//1-
   F460 : BOOL ;	//1-
   F461 : BOOL ;	//1-
   F462 : BOOL ;	//1-
   F463 : BOOL ;	//1-
   F464 : BOOL ;	//1-
   F465 : BOOL ;	//1-
   F466 : BOOL ;	//1-
   F467 : BOOL ;	//1-
   F468 : BOOL ;	//1-
   F469 : BOOL ;	//1-
   F470 : BOOL ;	//1-
   F471 : BOOL ;	//1-
   F472 : BOOL ;	//1-
   F473 : BOOL ;	//1-
   F474 : BOOL ;	//1-
   F475 : BOOL ;	//1-
   F476 : BOOL ;	//1-
   F477 : BOOL ;	//1-
   F478 : BOOL ;	//1-
   F479 : BOOL ;	//1-
   F480 : BOOL ;	//1-
   F481 : BOOL ;	//1-
   F482 : BOOL ;	//1-
   F483 : BOOL ;	//1-
   F484 : BOOL ;	//1-
   F485 : BOOL ;	//1-
   F486 : BOOL ;	//1-
   F487 : BOOL ;	//1-
   F488 : BOOL ;	//1-
   F489 : BOOL ;	//1-
   F490 : BOOL ;	//1-
   F491 : BOOL ;	//1-
   F492 : BOOL ;	//1-
   F493 : BOOL ;	//1-
   F494 : BOOL ;	//1-
   F495 : BOOL ;	//1-
   F496 : BOOL ;	//1-
   F497 : BOOL ;	//1-
   F498 : BOOL ;	//1-
   F499 : BOOL ;	//1-
   F500 : BOOL ;	//1-
   F501 : BOOL ;	//1-
   F502 : BOOL ;	//1-
   F503 : BOOL ;	//1-
   F504 : BOOL ;	//1-
   F505 : BOOL ;	//1-
   F506 : BOOL ;	//1-
   F507 : BOOL ;	//1-
   F508 : BOOL ;	//1-
   F509 : BOOL ;	//1-
   F510 : BOOL ;	//1-
   F511 : BOOL ;	//1-
   F512 : BOOL ;	//1-
   MSG_513 : BOOL ;	//Schaltschranktüre(n) an Werkzeugmaschine geöffnet
   MSG_514 : BOOL ;	//Schaltschranktüre(n) an Kühlschmierstoffanlage geöffnet
   MSG_515 : BOOL ;	//Schaltschranktemperatur zu hoch
   Me516 : BOOL ;	//1-
   Me517 : BOOL ;	//1-
   Me518 : BOOL ;	//1-
   Me519 : BOOL ;	//1-
   Me520 : BOOL ;	//1-
   Me521 : BOOL ;	//1-
   Me522 : BOOL ;	//1-
   Me523 : BOOL ;	//1-
   Me524 : BOOL ;	//1-
   Me525 : BOOL ;	//1-
   Me526 : BOOL ;	//1-
   Me527 : BOOL ;	//1-
   Me528 : BOOL ;	//1-
   Me529 : BOOL ;	//1-
   Me530 : BOOL ;	//1-
   Me531 : BOOL ;	//1-
   Me532 : BOOL ;	//1-
   Me533 : BOOL ;	//1-
   Me534 : BOOL ;	//1-
   Me535 : BOOL ;	//1-
   Me536 : BOOL ;	//1-
   Me537 : BOOL ;	//1-
   Me538 : BOOL ;	//1-
   Me539 : BOOL ;	//1-
   Me540 : BOOL ;	//1-
   Me541 : BOOL ;	//1-
   Me542 : BOOL ;	//1-
   Me543 : BOOL ;	//1-
   Me544 : BOOL ;	//1-
   Me545 : BOOL ;	//1-
   Me546 : BOOL ;	//1-
   Me547 : BOOL ;	//1-
   Me548 : BOOL ;	//1-
   Me549 : BOOL ;	//1-
   Me550 : BOOL ;	//1-
   Me551 : BOOL ;	//1-
   Me552 : BOOL ;	//1-
   Me553 : BOOL ;	//1-
   Me554 : BOOL ;	//1-
   Me555 : BOOL ;	//1-
   Me556 : BOOL ;	//1-
   Me557 : BOOL ;	//1-
   Me558 : BOOL ;	//1-
   Me559 : BOOL ;	//1-
   Me560 : BOOL ;	//1-
   MSG_561 : BOOL ;	//ext.Km-Anlage:Warnung steht an
   MSG_562 : BOOL ;	//Warnung:Kühlmittelfeinfilter verschmutzt E10.2
   MSG_563 : BOOL ;	//Druckvorgabe von LPlc nicht übernommen da nicht in Toleranz
   Me564 : BOOL ;	//1-
   Me565 : BOOL ;	//1-
   Me566 : BOOL ;	//1-
   Me567 : BOOL ;	//1-
   Me568 : BOOL ;	//1-
   Me569 : BOOL ;	//1-
   Me570 : BOOL ;	//1-
   Me571 : BOOL ;	//1-
   Me572 : BOOL ;	//1-
   Me573 : BOOL ;	//1-
   Me574 : BOOL ;	//1-
   Me575 : BOOL ;	//1-
   Me576 : BOOL ;	//1-
   Me577 : BOOL ;	//1-
   Me578 : BOOL ;	//1-
   Me579 : BOOL ;	//1-
   Me580 : BOOL ;	//1-
   Me581 : BOOL ;	//1-
   Me582 : BOOL ;	//1-
   Me583 : BOOL ;	//1-
   Me584 : BOOL ;	//1-
   Me585 : BOOL ;	//1-
   Me586 : BOOL ;	//1-
   Me587 : BOOL ;	//1-
   Me588 : BOOL ;	//1-
   Me589 : BOOL ;	//1-
   Me590 : BOOL ;	//1-
   Me591 : BOOL ;	//1-
   Me592 : BOOL ;	//1-
   Me593 : BOOL ;	//1-
   Me594 : BOOL ;	//1-
   Me595 : BOOL ;	//1-
   Me596 : BOOL ;	//1-
   Me597 : BOOL ;	//1-
   Me598 : BOOL ;	//1-
   Me599 : BOOL ;	//1-
   Me600 : BOOL ;	//1-
   Me601 : BOOL ;	//1-
   Me602 : BOOL ;	//1-
   Me603 : BOOL ;	//1-
   Me604 : BOOL ;	//1-
   Me605 : BOOL ;	//1-
   Me606 : BOOL ;	//1-
   Me607 : BOOL ;	//1-
   Me608 : BOOL ;	//1-
   Me609 : BOOL ;	//1-
   Me610 : BOOL ;	//1-
   Me611 : BOOL ;	//1-
   Me612 : BOOL ;	//1-
   Me613 : BOOL ;	//1-
   Me614 : BOOL ;	//1-
   Me615 : BOOL ;	//1-
   Me616 : BOOL ;	//1-
   Me617 : BOOL ;	//1-
   Me618 : BOOL ;	//1-
   Me619 : BOOL ;	//1-
   Me620 : BOOL ;	//1-
   Me621 : BOOL ;	//1-
   Me622 : BOOL ;	//1-
   Me623 : BOOL ;	//1-
   Me624 : BOOL ;	//1-
   Me625 : BOOL ;	//1-
   Me626 : BOOL ;	//1-
   Me627 : BOOL ;	//1-
   Me628 : BOOL ;	//1-
   Me629 : BOOL ;	//1-
   Me630 : BOOL ;	//1-
   Me631 : BOOL ;	//1-
   Me632 : BOOL ;	//1-
   Me633 : BOOL ;	//1-
   Me634 : BOOL ;	//1-
   Me635 : BOOL ;	//1-
   Me636 : BOOL ;	//1-
   Me637 : BOOL ;	//1-
   Me638 : BOOL ;	//1-
   Me639 : BOOL ;	//1-
   Me640 : BOOL ;	//1-
   Me641 : BOOL ;	//1-
   Me642 : BOOL ;	//1-
   Me643 : BOOL ;	//1-
   Me644 : BOOL ;	//1-
   Me645 : BOOL ;	//1-
   Me646 : BOOL ;	//1-
   Me647 : BOOL ;	//1-
   Me648 : BOOL ;	//1-
   Me649 : BOOL ;	//1-
   Me650 : BOOL ;	//1-
   Me651 : BOOL ;	//1-
   Me652 : BOOL ;	//1-
   Me653 : BOOL ;	//1-
   Me654 : BOOL ;	//1-
   Me655 : BOOL ;	//1-
   Me656 : BOOL ;	//1-
   Me657 : BOOL ;	//1-
   Me658 : BOOL ;	//1-
   Me659 : BOOL ;	//1-
   Me660 : BOOL ;	//1-
   Me661 : BOOL ;	//1-
   Me662 : BOOL ;	//1-
   Me663 : BOOL ;	//1-
   Me664 : BOOL ;	//1-
   Me665 : BOOL ;	//1-
   Me666 : BOOL ;	//1-
   Me667 : BOOL ;	//1-
   Me668 : BOOL ;	//1-
   Me669 : BOOL ;	//1-
   Me670 : BOOL ;	//1-
   Me671 : BOOL ;	//1-
   Me672 : BOOL ;	//1-
   Me673 : BOOL ;	//1-
   Me674 : BOOL ;	//1-
   Me675 : BOOL ;	//1-
   Me676 : BOOL ;	//1-
   Me677 : BOOL ;	//1-
   Me678 : BOOL ;	//1-
   Me679 : BOOL ;	//1-
   Me680 : BOOL ;	//1-
   Me681 : BOOL ;	//1-
   Me682 : BOOL ;	//1-
   Me683 : BOOL ;	//1-
   Me684 : BOOL ;	//1-
   Me685 : BOOL ;	//1-
   Me686 : BOOL ;	//1-
   Me687 : BOOL ;	//1-
   Me688 : BOOL ;	//1-
   Me689 : BOOL ;	//1-
   Me690 : BOOL ;	//1-
   Me691 : BOOL ;	//1-
   Me692 : BOOL ;	//1-
   Me693 : BOOL ;	//1-
   Me694 : BOOL ;	//1-
   Me695 : BOOL ;	//1-
   Me696 : BOOL ;	//1-
   Me697 : BOOL ;	//1-
   Me698 : BOOL ;	//1-
   Me699 : BOOL ;	//1-
   Me700 : BOOL ;	//1-
   Me701 : BOOL ;	//1-
   Me702 : BOOL ;	//1-
   Me703 : BOOL ;	//1-
   Me704 : BOOL ;	//1-
   Me705 : BOOL ;	//1-
   Me706 : BOOL ;	//1-
   Me707 : BOOL ;	//1-
   Me708 : BOOL ;	//1-
   Me709 : BOOL ;	//1-
   Me710 : BOOL ;	//1-
   Me711 : BOOL ;	//1-
   Me712 : BOOL ;	//1-
   Me713 : BOOL ;	//1-
   Me714 : BOOL ;	//1-
   Me715 : BOOL ;	//1-
   Me716 : BOOL ;	//1-
   Me717 : BOOL ;	//1-
   Me718 : BOOL ;	//1-
   Me719 : BOOL ;	//1-
   Me720 : BOOL ;	//1-
   Me721 : BOOL ;	//1-
   Me722 : BOOL ;	//1-
   Me723 : BOOL ;	//1-
   Me724 : BOOL ;	//1-
   Me725 : BOOL ;	//1-
   Me726 : BOOL ;	//1-
   Me727 : BOOL ;	//1-
   Me728 : BOOL ;	//1-
   Me729 : BOOL ;	//1-
   Me730 : BOOL ;	//1-
   Me731 : BOOL ;	//1-
   Me732 : BOOL ;	//1-
   Me733 : BOOL ;	//1-
   Me734 : BOOL ;	//1-
   Me735 : BOOL ;	//1-
   Me736 : BOOL ;	//1-
   Me737 : BOOL ;	//1-
   Me738 : BOOL ;	//1-
   Me739 : BOOL ;	//1-
   Me740 : BOOL ;	//1-
   Me741 : BOOL ;	//1-
   Me742 : BOOL ;	//1-
   Me743 : BOOL ;	//1-
   Me744 : BOOL ;	//1-
   Me745 : BOOL ;	//1-
   Me746 : BOOL ;	//1-
   Me747 : BOOL ;	//1-
   Me748 : BOOL ;	//1-
   Me749 : BOOL ;	//1-
   Me750 : BOOL ;	//1-
   Me751 : BOOL ;	//1-
   Me752 : BOOL ;	//1-
   Me753 : BOOL ;	//1-
   Me754 : BOOL ;	//1-
   Me755 : BOOL ;	//1-
   Me756 : BOOL ;	//1-
   Me757 : BOOL ;	//1-
   Me758 : BOOL ;	//1-
   Me759 : BOOL ;	//1-
   Me760 : BOOL ;	//1-
   Me761 : BOOL ;	//1-
   Me762 : BOOL ;	//1-
   Me763 : BOOL ;	//1-
   Me764 : BOOL ;	//1-
   Me765 : BOOL ;	//1-
   Me766 : BOOL ;	//1-
   Me767 : BOOL ;	//1-
   Me768 : BOOL ;	//1-
   Me769 : BOOL ;	//1-
   Me770 : BOOL ;	//1-
   Me771 : BOOL ;	//1-
   Me772 : BOOL ;	//1-
   Me773 : BOOL ;	//1-
   Me774 : BOOL ;	//1-
   Me775 : BOOL ;	//1-
   Me776 : BOOL ;	//1-
   Me777 : BOOL ;	//1-
   Me778 : BOOL ;	//1-
   Me779 : BOOL ;	//1-
   Me780 : BOOL ;	//1-
   Me781 : BOOL ;	//1-
   Me782 : BOOL ;	//1-
   Me783 : BOOL ;	//1-
   Me784 : BOOL ;	//1-
   Me785 : BOOL ;	//1-
   Me786 : BOOL ;	//1-
   Me787 : BOOL ;	//1-
   Me788 : BOOL ;	//1-
   Me789 : BOOL ;	//1-
   Me790 : BOOL ;	//1-
   Me791 : BOOL ;	//1-
   Me792 : BOOL ;	//1-
   Me793 : BOOL ;	//1-
   Me794 : BOOL ;	//1-
   Me795 : BOOL ;	//1-
   Me796 : BOOL ;	//1-
   Me797 : BOOL ;	//1-
   Me798 : BOOL ;	//1-
   Me799 : BOOL ;	//1-
   Me800 : BOOL ;	//1-
   Me801 : BOOL ;	//1-
   Me802 : BOOL ;	//1-
   Me803 : BOOL ;	//1-
   Me804 : BOOL ;	//1-
   Me805 : BOOL ;	//1-
   Me806 : BOOL ;	//1-
   Me807 : BOOL ;	//1-
   Me808 : BOOL ;	//1-
   Me809 : BOOL ;	//1-
   Me810 : BOOL ;	//1-
   Me811 : BOOL ;	//1-
   Me812 : BOOL ;	//1-
   Me813 : BOOL ;	//1-
   Me814 : BOOL ;	//1-
   Me815 : BOOL ;	//1-
   Me816 : BOOL ;	//1-
   Me817 : BOOL ;	//1-
   Me818 : BOOL ;	//1-
   Me819 : BOOL ;	//1-
   Me820 : BOOL ;	//1-
   Me821 : BOOL ;	//1-
   Me822 : BOOL ;	//1-
   Me823 : BOOL ;	//1-
   Me824 : BOOL ;	//1-
   Me825 : BOOL ;	//1-
   Me826 : BOOL ;	//1-
   Me827 : BOOL ;	//1-
   Me828 : BOOL ;	//1-
   Me829 : BOOL ;	//1-
   Me830 : BOOL ;	//1-
   Me831 : BOOL ;	//1-
   Me832 : BOOL ;	//1-
   Me833 : BOOL ;	//1-
   Me834 : BOOL ;	//1-
   Me835 : BOOL ;	//1-
   Me836 : BOOL ;	//1-
   Me837 : BOOL ;	//1-
   Me838 : BOOL ;	//1-
   Me839 : BOOL ;	//1-
   Me840 : BOOL ;	//1-
   Me841 : BOOL ;	//1-
   Me842 : BOOL ;	//1-
   Me843 : BOOL ;	//1-
   Me844 : BOOL ;	//1-
   Me845 : BOOL ;	//1-
   Me846 : BOOL ;	//1-
   Me847 : BOOL ;	//1-
   Me848 : BOOL ;	//1-
   Me849 : BOOL ;	//1-
   Me850 : BOOL ;	//1-
   Me851 : BOOL ;	//1-
   Me852 : BOOL ;	//1-
   Me853 : BOOL ;	//1-
   Me854 : BOOL ;	//1-
   Me855 : BOOL ;	//1-
   Me856 : BOOL ;	//1-
   Me857 : BOOL ;	//1-
   Me858 : BOOL ;	//1-
   Me859 : BOOL ;	//1-
   Me860 : BOOL ;	//1-
   Me861 : BOOL ;	//1-
   Me862 : BOOL ;	//1-
   Me863 : BOOL ;	//1-
   Me864 : BOOL ;	//1-
   Me865 : BOOL ;	//1-
   Me866 : BOOL ;	//1-
   Me867 : BOOL ;	//1-
   Me868 : BOOL ;	//1-
   Me869 : BOOL ;	//1-
   Me870 : BOOL ;	//1-
   Me871 : BOOL ;	//1-
   Me872 : BOOL ;	//1-
   Me873 : BOOL ;	//1-
   Me874 : BOOL ;	//1-
   Me875 : BOOL ;	//1-
   Me876 : BOOL ;	//1-
   Me877 : BOOL ;	//1-
   Me878 : BOOL ;	//1-
   Me879 : BOOL ;	//1-
   Me880 : BOOL ;	//1-
   Me881 : BOOL ;	//1-
   Me882 : BOOL ;	//1-
   Me883 : BOOL ;	//1-
   Me884 : BOOL ;	//1-
   Me885 : BOOL ;	//1-
   Me886 : BOOL ;	//1-
   Me887 : BOOL ;	//1-
   Me888 : BOOL ;	//1-
   Me889 : BOOL ;	//1-
   Me890 : BOOL ;	//1-
   Me891 : BOOL ;	//1-
   Me892 : BOOL ;	//1-
   Me893 : BOOL ;	//1-
   Me894 : BOOL ;	//1-
   Me895 : BOOL ;	//1-
   Me896 : BOOL ;	//1-
   Me897 : BOOL ;	//1-
   Me898 : BOOL ;	//1-
   Me899 : BOOL ;	//1-
   Me900 : BOOL ;	//1-
   Me901 : BOOL ;	//1-
   Me902 : BOOL ;	//1-
   Me903 : BOOL ;	//1-
   Me904 : BOOL ;	//1-
   Me905 : BOOL ;	//1-
   Me906 : BOOL ;	//1-
   Me907 : BOOL ;	//1-
   Me908 : BOOL ;	//1-
   Me909 : BOOL ;	//1-
   Me910 : BOOL ;	//1-
   Me911 : BOOL ;	//1-
   Me912 : BOOL ;	//1-
   Me913 : BOOL ;	//1-
   Me914 : BOOL ;	//1-
   Me915 : BOOL ;	//1-
   Me916 : BOOL ;	//1-
   Me917 : BOOL ;	//1-
   Me918 : BOOL ;	//1-
   Me919 : BOOL ;	//1-
   Me920 : BOOL ;	//1-
   Me921 : BOOL ;	//1-
   Me922 : BOOL ;	//1-
   Me923 : BOOL ;	//1-
   Me924 : BOOL ;	//1-
   Me925 : BOOL ;	//1-
   Me926 : BOOL ;	//1-
   Me927 : BOOL ;	//1-
   Me928 : BOOL ;	//1-
   Me929 : BOOL ;	//1-
   Me930 : BOOL ;	//1-
   Me931 : BOOL ;	//1-
   Me932 : BOOL ;	//1-
   Me933 : BOOL ;	//1-
   Me934 : BOOL ;	//1-
   Me935 : BOOL ;	//1-
   Me936 : BOOL ;	//1-
   Me937 : BOOL ;	//1-
   Me938 : BOOL ;	//1-
   Me939 : BOOL ;	//1-
   Me940 : BOOL ;	//1-
   Me941 : BOOL ;	//1-
   Me942 : BOOL ;	//1-
   Me943 : BOOL ;	//1-
   Me944 : BOOL ;	//1-
   Me945 : BOOL ;	//1-
   Me946 : BOOL ;	//1-
   Me947 : BOOL ;	//1-
   Me948 : BOOL ;	//1-
   Me949 : BOOL ;	//1-
   Me950 : BOOL ;	//1-
   Me951 : BOOL ;	//1-
   Me952 : BOOL ;	//1-
   Me953 : BOOL ;	//1-
   Me954 : BOOL ;	//1-
   Me955 : BOOL ;	//1-
   Me956 : BOOL ;	//1-
   Me957 : BOOL ;	//1-
   Me958 : BOOL ;	//1-
   Me959 : BOOL ;	//1-
   Me960 : BOOL ;	//1-
   Me961 : BOOL ;	//1-
   Me962 : BOOL ;	//1-
   Me963 : BOOL ;	//1-
   Me964 : BOOL ;	//1-
   Me965 : BOOL ;	//1-
   Me966 : BOOL ;	//1-
   Me967 : BOOL ;	//1-
   Me968 : BOOL ;	//1-
   Me969 : BOOL ;	//1-
   Me970 : BOOL ;	//1-
   Me971 : BOOL ;	//1-
   Me972 : BOOL ;	//1-
   Me973 : BOOL ;	//1-
   Me974 : BOOL ;	//1-
   Me975 : BOOL ;	//1-
   Me976 : BOOL ;	//1-
   Me977 : BOOL ;	//1-
   Me978 : BOOL ;	//1-
   Me979 : BOOL ;	//1-
   Me980 : BOOL ;	//1-
   Me981 : BOOL ;	//1-
   Me982 : BOOL ;	//1-
   Me983 : BOOL ;	//1-
   Me984 : BOOL ;	//1-
   Me985 : BOOL ;	//1-
   Me986 : BOOL ;	//1-
   Me987 : BOOL ;	//1-
   Me988 : BOOL ;	//1-
   Me989 : BOOL ;	//1-
   Me990 : BOOL ;	//1-
   Me991 : BOOL ;	//1-
   Me992 : BOOL ;	//1-
   Me993 : BOOL ;	//1-
   Me994 : BOOL ;	//1-
   Me995 : BOOL ;	//1-
   Me996 : BOOL ;	//1-
   Me997 : BOOL ;	//1-
   Me998 : BOOL ;	//1-
   Me999 : BOOL ;	//1-
   Me1000 : BOOL ;	//1-
   Me1001 : BOOL ;	//1-
   Me1002 : BOOL ;	//1-
   Me1003 : BOOL ;	//1-
   Me1004 : BOOL ;	//1-
   Me1005 : BOOL ;	//1-
   Me1006 : BOOL ;	//1-
   Me1007 : BOOL ;	//1-
   Me1008 : BOOL ;	//1-
   Me1009 : BOOL ;	//1-
   Me1010 : BOOL ;	//1-
   Me1011 : BOOL ;	//1-
   Me1012 : BOOL ;	//1-
   Me1013 : BOOL ;	//1-
   Me1014 : BOOL ;	//1-
   Me1015 : BOOL ;	//1-
   Me1016 : BOOL ;	//1-
   Me1017 : BOOL ;	//1-
   Me1018 : BOOL ;	//1-
   Me1019 : BOOL ;	//1-
   Me1020 : BOOL ;	//1-
   Me1021 : BOOL ;	//1-
   Me1022 : BOOL ;	//1-
   Me1023 : BOOL ;	//1-
   Me1024 : BOOL ;	//1-
  END_STRUCT ;	
END_TYPE

TYPE "UDT_COOLANT"	// UDT 50
VERSION : 0.1
  STRUCT
   PSoll : INT ;	//stat:letzter gespeicherter KmSolldruck
   PSollAlt : INT ;	//stat:letzter gespeich.KmSolldruck (alt, für Änderungserfassung)
   PSollAA : INT ;	//stat:letzter gespeich.KmSolldruck, berechnet für AA
   P20AA : INT ;	//stat:Solldruck 20Bar, berechnet für AA
   P40AA : INT ;	//stat:Solldruck 40Bar, berechnet für AA
   fk : ARRAY  [0 .. 15 ] OF //stat:Flankenhilfsmerker
   BOOL ;
   hvFEin : BOOL ;	//stat:KmHauptventil Fehler:Einschaltüberwachung
   hvFUnt : BOOL ;	//stat:KmHauptventil Fehler:Unterbrechungsüberwachung
   kmdFEin : BOOL ;	//stat:KmSystem=Niederdruck Fehler:Einschaltüberwachung
   kmdFUnt : BOOL ;	//stat:KmSystem=Niederdruck Fehler:Unterbrechungsüberwachung
   FlFEin : BOOL ;	//stat:KmDurchfluss Fehler:Einschaltüberwachung
   FlFUnt : BOOL ;	//stat:KmDurchfluss Fehler:Unterbrechungsüberwachung
   x6 : BOOL ;
   x7 : BOOL ;
   x8 : BOOL ;
   x9 : BOOL ;
   x10 : BOOL ;
   x11 : BOOL ;
   x12 : BOOL ;
   x13 : BOOL ;
   x14 : BOOL ;
   x15 : BOOL ;
  END_STRUCT ;	
END_TYPE

TYPE "UDT101"	// UDT 101
AUTHOR : SPAC_slh
VERSION : 0.1
  STRUCT
   T : ARRAY  [0 .. 31 ] OF UDT 1010;
  END_STRUCT ;	
END_TYPE

TYPE "UDT1010"	// UDT 1010
AUTHOR : SPAC_slh
VERSION : 0.1
  STRUCT
   SwT : ARRAY  [0 .. 2 ] OF //SwZeit[0]
   TIME ;
   x : STRUCT
    E1gs : BOOL ;	//Endlage 1 gespeichert
    E2gs : BOOL ;	//Endlage 2 gespeichert
    x2 : BOOL ;
    x3 : BOOL ;
    x4 : BOOL ;
    x5 : BOOL ;
    x6 : BOOL ;
    x7 : BOOL ;
    fk0 : BOOL ;
    fk1 : BOOL ;
    fk2 : BOOL ;
    fk3 : BOOL ;
    fk4 : BOOL ;
    fk5 : BOOL ;
    fk6 : BOOL ;
    fk7 : BOOL ;
   END_STRUCT ;
  END_STRUCT ;	
END_TYPE

FUNCTION_BLOCK "TOOLING SYSTEM???"	// FB 15
AUTHOR : A.Petz
VERSION : 0.4
BEGIN
// (block stored without names or comments; labels and parameter names are numbered)
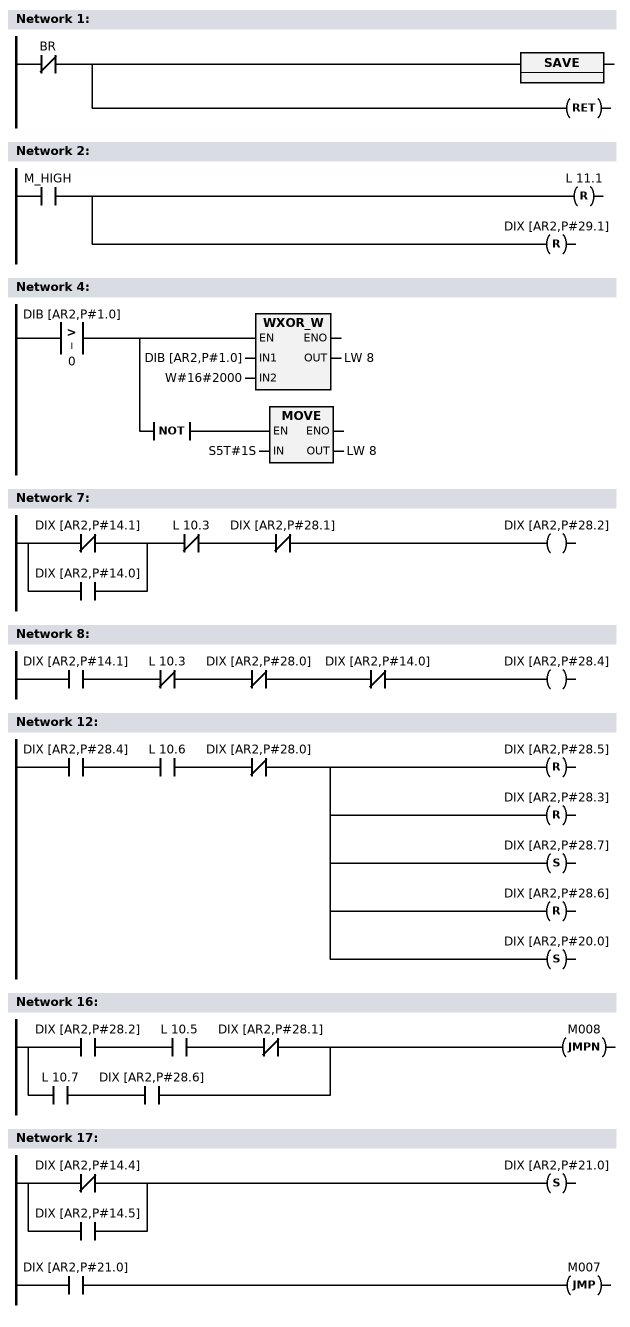
NETWORK
TITLE =
      AN    BR;
      SAVE;
      BEC;
NETWORK
TITLE =
      A     "M_HIGH";
      R     L 11.1;
      R     DIX [AR2,P#29.1];
NETWORK
TITLE =
      L     DIB [AR2,P#0.0];
      CAW;
      TAR1  LD 0;
      LAR1  P#L 6.0;
      T     LW [AR1,P#0.0];
      LAR1  LD 0;
NETWORK
TITLE =
      L     DIB [AR2,P#1.0];
      L     0;
      >I;
      =     L 12.0;
      A     L 12.0;
      JNB   M001;
      L     DIB [AR2,P#1.0];
      L     W#16#2000;
      XOW;
      T     LW 8;
M001: NOP   0;
      A     L 12.0;
      NOT;
      JNB   M002;
      L     S5T#1S;
      T     LW 8;
M002: NOP   0;
NETWORK
TITLE =
      A     "M_HIGH";
      =     L 10.2;
NETWORK
TITLE =
      O(;
      L     DB2.DBW 2;
      L     0;
      <>I;
      );
      O     "DB_MESSAGE".F033;
      O     "DB_MESSAGE".F034;
      O     "DB_MESSAGE".F035;
      O     "DB_MESSAGE".F036;
      =     L 10.3;
NETWORK
TITLE =
      A(;
      ON    DIX [AR2,P#14.1];
      O     DIX [AR2,P#14.0];
      );
      AN    L 10.3;
      AN    DIX [AR2,P#28.1];
      =     DIX [AR2,P#28.2];
NETWORK
TITLE =
      A     DIX [AR2,P#14.1];
      AN    L 10.3;
      AN    DIX [AR2,P#28.0];
      AN    DIX [AR2,P#14.0];
      =     DIX [AR2,P#28.4];
NETWORK
TITLE =
      A     DIX [AR2,P#28.2];
      FP    DIX [AR2,P#26.0];
      =     L 10.5;
      A     L 10.5;
      O(;
      A     DIX [AR2,P#28.4];
      FP    DIX [AR2,P#26.1];
      =     L 10.6;
      A     L 10.6;
      );
      O(;
      A     L 10.3;
      FN    DIX [AR2,P#26.2];
      =     L 10.7;
      A     L 10.7;
      );
      O     DIX [AR2,P#15.3];
      =     L 10.1;
NETWORK
TITLE =
      AN    L 10.1;
      JC    M003;
      TAR1  LD 0;
      LAR1  P#DIX 20.0;
      L     0;
      T     DIW [AR1,P#0.0];
      LAR1  LD 0;
M003: NOP   0;
NETWORK
TITLE =
      A(;
      A     DIX [AR2,P#15.5];
      AN    DIX [AR2,P#15.6];
      O     DIX [AR2,P#14.0];
      );
      =     L 10.1;
      A     L 10.1;
      A     L 10.5;
      S     DIX [AR2,P#29.0];
      AN    L 10.1;
      A     L 10.5;
      R     DIX [AR2,P#29.0];
      NOP   0;
NETWORK
TITLE =
      A     DIX [AR2,P#28.4];
      A     L 10.6;
      AN    DIX [AR2,P#28.0];
      R     DIX [AR2,P#28.5];
      R     DIX [AR2,P#28.3];
      S     DIX [AR2,P#28.7];
      R     DIX [AR2,P#28.6];
      S     DIX [AR2,P#20.0];
NETWORK
TITLE =
      A     DIX [AR2,P#28.4];
      A     DIX [AR2,P#20.0];
      =     L 12.0;
      A     L 12.0;
      A(;
      T     LD 13;
      TAK;
      T     LD 17;
      L     DIW [AR2,P#2.0];
      T     LW 21;
      L     LD 17;
      L     LD 13;
      O     T [LW 21];
      ON    L 6.0;
      );
      R     DIX [AR2,P#20.0];
      S     DIX [AR2,P#20.1];
      S     L 11.1;
      A     L 12.0;
      BLD   102;
      S     DIX [AR2,P#29.1];
      A     L 12.0;
      JNB   M004;
      L     LW 8;
      T     DIW [AR2,P#18.0];
M004: NOP   0;
NETWORK
TITLE =
      A     DIX [AR2,P#28.4];
      A     DIX [AR2,P#20.1];
      A     DIX [AR2,P#22.1];
      =     L 12.0;
      A     L 12.0;
      T     LD 13;
      TAK;
      T     LD 17;
      L     DIW [AR2,P#2.0];
      T     LW 21;
      L     LD 17;
      L     LD 13;
      A     T [LW 21];
      R     DIX [AR2,P#20.1];
      S     DIX [AR2,P#20.2];
      S     L 11.1;
      A     L 12.0;
      BLD   102;
      S     DIX [AR2,P#29.1];
      A     L 12.0;
      JNB   M005;
      L     S5T#3S;
      T     DIW [AR2,P#18.0];
M005: NOP   0;
NETWORK
TITLE =
      A     DIX [AR2,P#28.4];
      A     DIX [AR2,P#20.2];
      A     DIX [AR2,P#22.2];
      =     L 12.0;
      A     L 12.0;
      T     LD 13;
      TAK;
      T     LD 17;
      L     DIW [AR2,P#2.0];
      T     LW 21;
      L     LD 17;
      L     LD 13;
      A     T [LW 21];
      R     DIX [AR2,P#20.2];
      R     DIX [AR2,P#28.7];
      S     DIX [AR2,P#28.5];
      S     L 11.1;
      A     L 12.0;
      BLD   102;
      S     DIX [AR2,P#29.1];
      A     L 12.0;
      JNB   M006;
      L     S5T#100MS;
      T     DIW [AR2,P#18.0];
M006: NOP   0;
NETWORK
TITLE =
      A     DIX [AR2,P#28.2];
      A     L 10.5;
      AN    DIX [AR2,P#28.1];
      O;
      A     L 10.7;
      A     DIX [AR2,P#28.6];
      JCN   M008;
NETWORK
TITLE =
      A(;
      ON    DIX [AR2,P#14.4];
      O     DIX [AR2,P#14.5];
      );
      S     DIX [AR2,P#21.0];
      NOP   0;
      A     DIX [AR2,P#21.0];
      JC    M007;
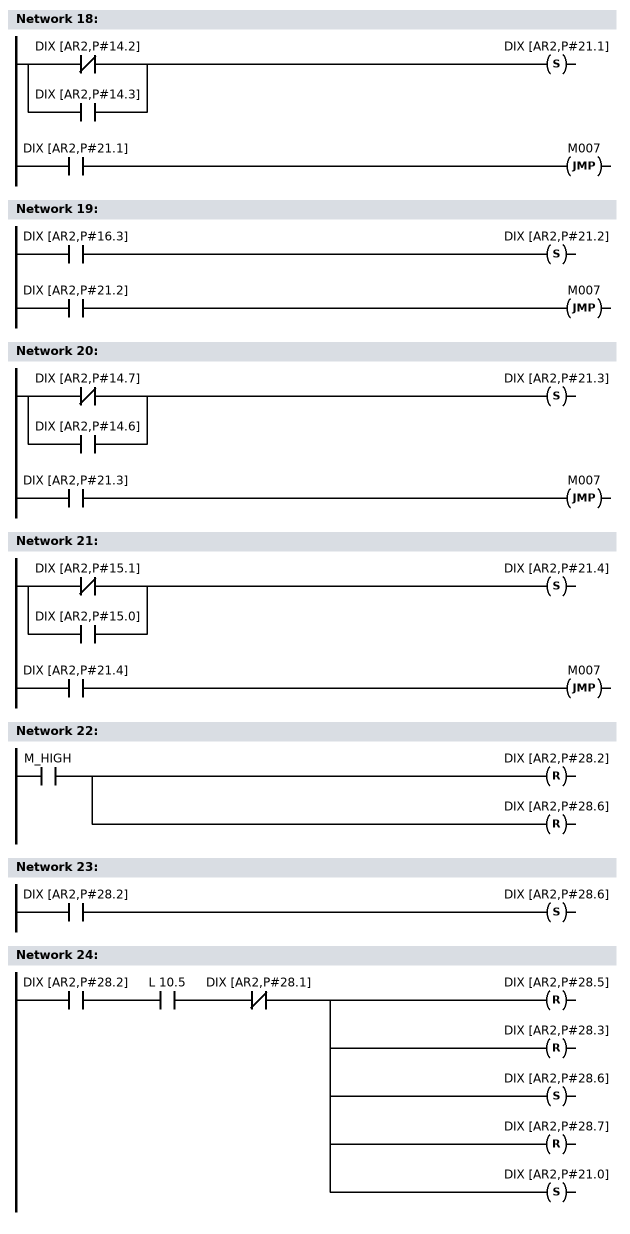
NETWORK
TITLE =
      A(;
      ON    DIX [AR2,P#14.2];
      O     DIX [AR2,P#14.3];
      );
      S     DIX [AR2,P#21.1];
      NOP   0;
      A     DIX [AR2,P#21.1];
      JC    M007;
NETWORK
TITLE =
      A     DIX [AR2,P#16.3];
      S     DIX [AR2,P#21.2];
      NOP   0;
      A     DIX [AR2,P#21.2];
      JC    M007;
NETWORK
TITLE =
      A(;
      ON    DIX [AR2,P#14.7];
      O     DIX [AR2,P#14.6];
      );
      S     DIX [AR2,P#21.3];
      NOP   0;
      A     DIX [AR2,P#21.3];
      JC    M007;
NETWORK
TITLE =
      A(;
      ON    DIX [AR2,P#15.1];
      O     DIX [AR2,P#15.0];
      );
      S     DIX [AR2,P#21.4];
      NOP   0;
      A     DIX [AR2,P#21.4];
      JC    M007;
NETWORK
TITLE =
      A     "M_HIGH";
      R     DIX [AR2,P#28.2];
      R     DIX [AR2,P#28.6];
NETWORK
TITLE =
M007: A     DIX [AR2,P#28.2];
      S     DIX [AR2,P#28.6];
NETWORK
TITLE =
M008: A     DIX [AR2,P#28.2];
      A     L 10.5;
      AN    DIX [AR2,P#28.1];
      R     DIX [AR2,P#28.5];
      R     DIX [AR2,P#28.3];
      S     DIX [AR2,P#28.6];
      R     DIX [AR2,P#28.7];
      S     DIX [AR2,P#21.0];
NETWORK
TITLE =
      A     DIX [AR2,P#28.2];
      A     DIX [AR2,P#21.0];
      A     DIX [AR2,P#23.0];
      =     L 12.0;
      A     L 12.0;
      T     LD 13;
      TAK;
      T     LD 17;
      L     DIW [AR2,P#2.0];
      T     LW 21;
      L     LD 17;
      L     LD 13;
      A     T [LW 21];
      R     DIX [AR2,P#21.0];
      S     DIX [AR2,P#21.1];
      S     L 11.1;
      A     L 12.0;
      BLD   102;
      S     DIX [AR2,P#29.1];
      A     L 12.0;
      JNB   M009;
      L     S5T#3S;
      T     DIW [AR2,P#18.0];
M009: NOP   0;
NETWORK
TITLE =
      A     DIX [AR2,P#28.2];
      A     DIX [AR2,P#21.1];
      A     DIX [AR2,P#23.1];
      =     L 12.0;
      A     L 12.0;
      T     LD 13;
      TAK;
      T     LD 17;
      L     DIW [AR2,P#2.0];
      T     LW 21;
      L     LD 17;
      L     LD 13;
      A     T [LW 21];
      R     DIX [AR2,P#21.1];
      S     DIX [AR2,P#21.2];
      S     L 11.1;
      A     L 12.0;
      BLD   102;
      S     DIX [AR2,P#29.1];
      A     L 12.0;
      JNB   M010;
      L     S5T#3S;
      T     DIW [AR2,P#18.0];
M010: NOP   0;
NETWORK
TITLE =
      A     DIX [AR2,P#28.2];
      A     DIX [AR2,P#21.2];
      A(;
      O     DIX [AR2,P#23.2];
      ON    L 6.0;
      );
      =     L 12.0;
      A     L 12.0;
      A(;
      T     LD 13;
      TAK;
      T     LD 17;
      L     DIW [AR2,P#2.0];
      T     LW 21;
      L     LD 17;
      L     LD 13;
      O     T [LW 21];
      ON    L 6.0;
      ON    L 6.1;
      O     DIX [AR2,P#29.0];
      );
      R     DIX [AR2,P#21.2];
      S     DIX [AR2,P#21.3];
      S     L 11.1;
      A     L 12.0;
      A     L 6.1;
      AN    DIX [AR2,P#29.0];
      =     L 12.1;
      A     L 12.1;
      BLD   102;
      S     DIX [AR2,P#29.1];
      A     L 12.1;
      JNB   M011;
      L     S5T#5S;
      T     DIW [AR2,P#18.0];
M011: NOP   0;
NETWORK
TITLE =
      A     DIX [AR2,P#28.2];
      A     DIX [AR2,P#21.3];
      A(;
      O     DIX [AR2,P#23.3];
      ON    L 6.1;
      O     DIX [AR2,P#29.0];
      );
      =     L 12.0;
      A     L 12.0;
      A(;
      T     LD 13;
      TAK;
      T     LD 17;
      L     DIW [AR2,P#2.0];
      T     LW 21;
      L     LD 17;
      L     LD 13;
      O     T [LW 21];
      ON    L 6.1;
      O     DIX [AR2,P#29.0];
      );
      R     DIX [AR2,P#21.3];
      S     DIX [AR2,P#21.4];
      S     L 11.1;
      A     L 12.0;
      BLD   102;
      S     DIX [AR2,P#29.1];
      A     L 12.0;
      JNB   M012;
      L     S5T#5S;
      T     DIW [AR2,P#18.0];
M012: NOP   0;
NETWORK
TITLE =
      A     DIX [AR2,P#28.2];
      A     DIX [AR2,P#21.4];
      A(;
      O     DIX [AR2,P#23.4];
      ON    L 6.2;
      O     DIX [AR2,P#29.0];
      );
      =     L 12.0;
      A     L 12.0;
      A(;
      T     LD 13;
      TAK;
      T     LD 17;
      L     DIW [AR2,P#2.0];
      T     LW 21;
      L     LD 17;
      L     LD 13;
      O     T [LW 21];
      ON    L 6.2;
      O     DIX [AR2,P#29.0];
      );
      R     DIX [AR2,P#21.4];
      S     DIX [AR2,P#28.3];
      R     DIX [AR2,P#28.6];
      A     L 12.0;
      BLD   102;
      S     DIX [AR2,P#29.1];
      A     L 12.0;
      JNB   M013;
      L     S5T#100MS;
      T     DIW [AR2,P#18.0];
M013: NOP   0;
NETWORK
TITLE =
      A     DIX [AR2,P#29.1];
      AN    L 11.1;
      L     DIW [AR2,P#18.0];
      T     LD 12;
      TAK;
      T     LD 16;
      L     DIW [AR2,P#2.0];
      T     LW 20;
      L     LD 16;
      L     LD 12;
      SD    T [LW 20];
NETWORK
TITLE =
      A     L 10.2;
      =     L 12.0;
      A     L 12.0;
      A(;
      A     DIX [AR2,P#20.1];
      A     DIX [AR2,P#28.4];
      O     DIX [AR2,P#22.1];
      );
      =     DIX [AR2,P#16.1];
      R     DIX [AR2,P#23.1];
      A     L 12.0;
      A(;
      A     DIX [AR2,P#21.1];
      A     DIX [AR2,P#28.2];
      O     DIX [AR2,P#23.1];
      );
      =     L 11.3;
      R     DIX [AR2,P#22.1];
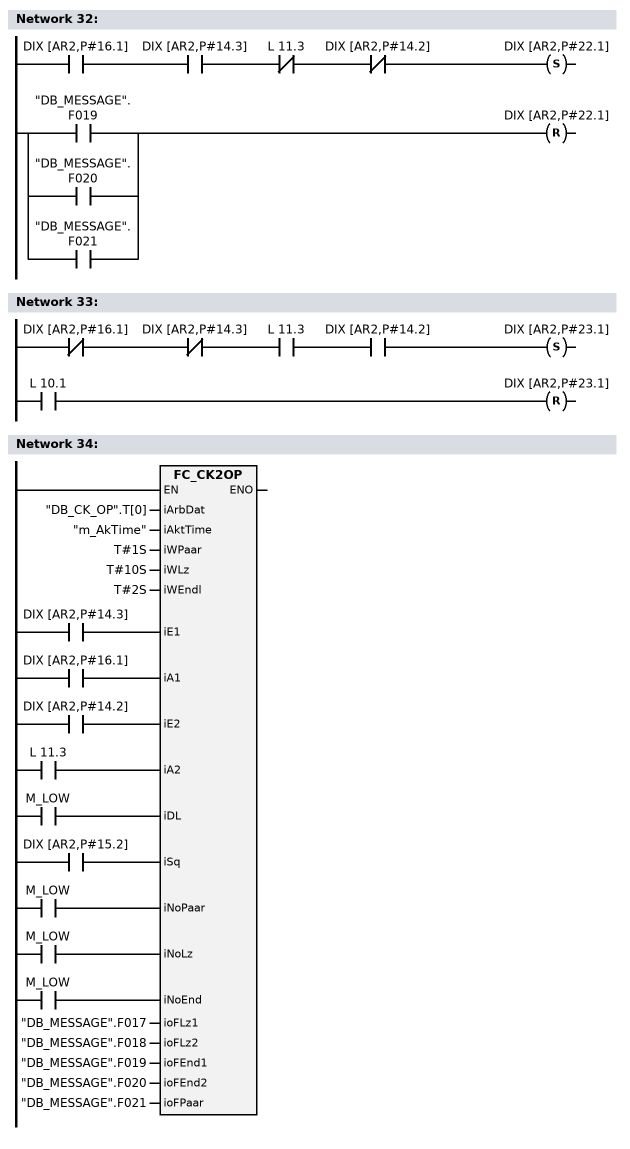
NETWORK
TITLE =
      A     DIX [AR2,P#16.1];
      A     DIX [AR2,P#14.3];
      AN    L 11.3;
      AN    DIX [AR2,P#14.2];
      S     DIX [AR2,P#22.1];
      A(;
      O     "DB_MESSAGE".F019;
      O     "DB_MESSAGE".F020;
      O     "DB_MESSAGE".F021;
      );
      =     L 10.1;
      A     L 10.1;
      R     DIX [AR2,P#22.1];
      NOP   0;
NETWORK
TITLE =
      AN    DIX [AR2,P#16.1];
      AN    DIX [AR2,P#14.3];
      A     L 11.3;
      A     DIX [AR2,P#14.2];
      S     DIX [AR2,P#23.1];
      A     L 10.1;
      R     DIX [AR2,P#23.1];
      NOP   0;
NETWORK
TITLE =
      A     DIX [AR2,P#14.3];
      =     L 12.0;
      BLD   103;
      A     DIX [AR2,P#16.1];
      =     L 12.1;
      BLD   103;
      A     DIX [AR2,P#14.2];
      =     L 12.2;
      BLD   103;
      A     L 11.3;
      =     L 12.3;
      BLD   103;
      A     "M_LOW";
      =     L 12.4;
      BLD   103;
      A     DIX [AR2,P#15.2];
      =     L 12.5;
      BLD   103;
      A     "M_LOW";
      =     L 12.6;
      BLD   103;
      A     "M_LOW";
      =     L 12.7;
      BLD   103;
      A     "M_LOW";
      =     L 13.0;
      BLD   103;
      CALL  "FC_CK2OP" (
           iArbDat                  := "DB_CK_OP".T[0],
           iAktTime                 := "m_AkTime",
           iWPaar                   := T#1S,
           iWLz                     := T#10S,
           iWEndl                   := T#2S,
           iE1                      := L 12.0,
           iA1                      := L 12.1,
           iE2                      := L 12.2,
           iA2                      := L 12.3,
           iDL                      := L 12.4,
           iSq                      := L 12.5,
           iNoPaar                  := L 12.6,
           iNoLz                    := L 12.7,
           iNoEnd                   := L 13.0,
           ioFLz1                   := "DB_MESSAGE".F017,
           ioFLz2                   := "DB_MESSAGE".F018,
           ioFEnd1                  := "DB_MESSAGE".F019,
           ioFEnd2                  := "DB_MESSAGE".F020,
           ioFPaar                  := "DB_MESSAGE".F021);
      NOP   0;
NETWORK
TITLE =
      A     L 10.2;
      =     L 12.0;
      A     L 12.0;
      A(;
      A     DIX [AR2,P#20.2];
      A     DIX [AR2,P#28.4];
      O     DIX [AR2,P#22.2];
      );
      =     DIX [AR2,P#16.2];
      R     DIX [AR2,P#23.0];
      A     L 12.0;
      A(;
      A     DIX [AR2,P#21.0];
      A     DIX [AR2,P#28.2];
      O     DIX [AR2,P#23.0];
      );
      =     L 11.4;
      R     DIX [AR2,P#22.2];
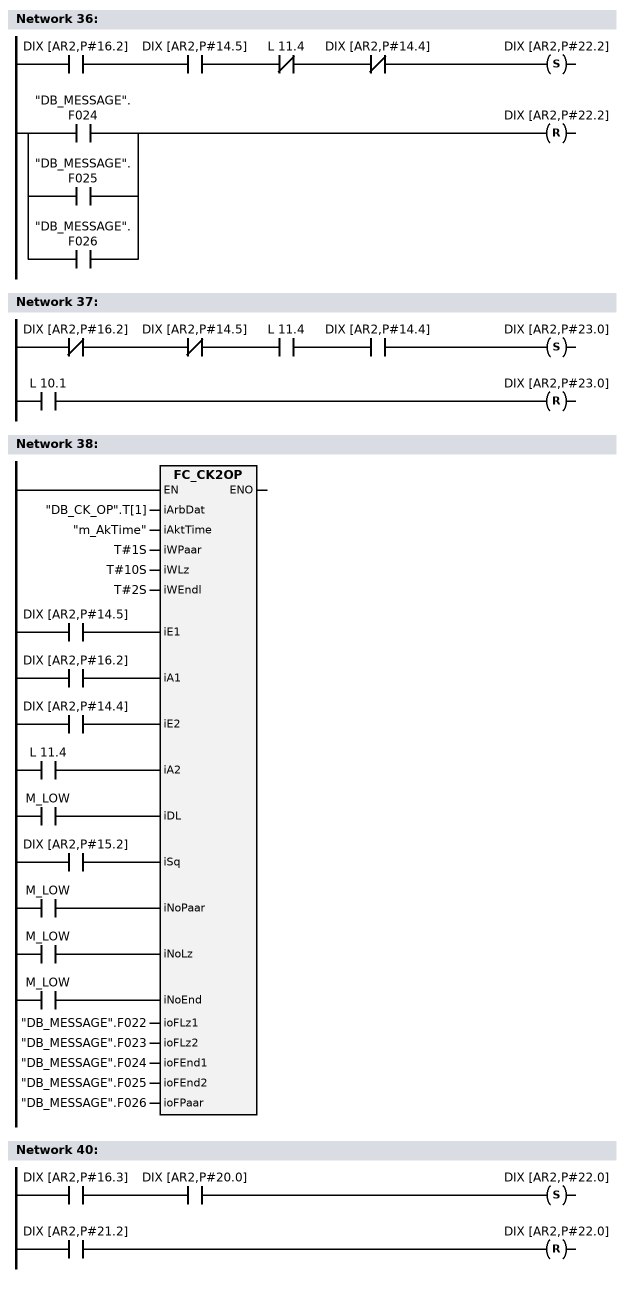
NETWORK
TITLE =
      A     DIX [AR2,P#16.2];
      A     DIX [AR2,P#14.5];
      AN    L 11.4;
      AN    DIX [AR2,P#14.4];
      S     DIX [AR2,P#22.2];
      A(;
      O     "DB_MESSAGE".F024;
      O     "DB_MESSAGE".F025;
      O     "DB_MESSAGE".F026;
      );
      =     L 10.1;
      A     L 10.1;
      R     DIX [AR2,P#22.2];
      NOP   0;
NETWORK
TITLE =
      AN    DIX [AR2,P#16.2];
      AN    DIX [AR2,P#14.5];
      A     L 11.4;
      A     DIX [AR2,P#14.4];
      S     DIX [AR2,P#23.0];
      A     L 10.1;
      R     DIX [AR2,P#23.0];
      NOP   0;
NETWORK
TITLE =
      A     DIX [AR2,P#14.5];
      =     L 12.0;
      BLD   103;
      A     DIX [AR2,P#16.2];
      =     L 12.1;
      BLD   103;
      A     DIX [AR2,P#14.4];
      =     L 12.2;
      BLD   103;
      A     L 11.4;
      =     L 12.3;
      BLD   103;
      A     "M_LOW";
      =     L 12.4;
      BLD   103;
      A     DIX [AR2,P#15.2];
      =     L 12.5;
      BLD   103;
      A     "M_LOW";
      =     L 12.6;
      BLD   103;
      A     "M_LOW";
      =     L 12.7;
      BLD   103;
      A     "M_LOW";
      =     L 13.0;
      BLD   103;
      CALL  "FC_CK2OP" (
           iArbDat                  := "DB_CK_OP".T[1],
           iAktTime                 := "m_AkTime",
           iWPaar                   := T#1S,
           iWLz                     := T#10S,
           iWEndl                   := T#2S,
           iE1                      := L 12.0,
           iA1                      := L 12.1,
           iE2                      := L 12.2,
           iA2                      := L 12.3,
           iDL                      := L 12.4,
           iSq                      := L 12.5,
           iNoPaar                  := L 12.6,
           iNoLz                    := L 12.7,
           iNoEnd                   := L 13.0,
           ioFLz1                   := "DB_MESSAGE".F022,
           ioFLz2                   := "DB_MESSAGE".F023,
           ioFEnd1                  := "DB_MESSAGE".F024,
           ioFEnd2                  := "DB_MESSAGE".F025,
           ioFPaar                  := "DB_MESSAGE".F026);
      NOP   0;
NETWORK
TITLE =
      A     L 10.2;
      AN    L 10.3;
      =     L 12.0;
      A     L 12.0;
      A(;
      A     DIX [AR2,P#20.0];
      A     DIX [AR2,P#28.4];
      O     DIX [AR2,P#22.0];
      );
      =     DIX [AR2,P#16.3];
      R     DIX [AR2,P#23.2];
      A     L 12.0;
      A(;
      A     DIX [AR2,P#21.2];
      A     DIX [AR2,P#28.2];
      O     DIX [AR2,P#23.2];
      );
      =     L 11.5;
      R     DIX [AR2,P#22.0];
NETWORK
TITLE =
      A     DIX [AR2,P#16.3];
      A     DIX [AR2,P#20.0];
      S     DIX [AR2,P#22.0];
      A     DIX [AR2,P#21.2];
      R     DIX [AR2,P#22.0];
      NOP   0;
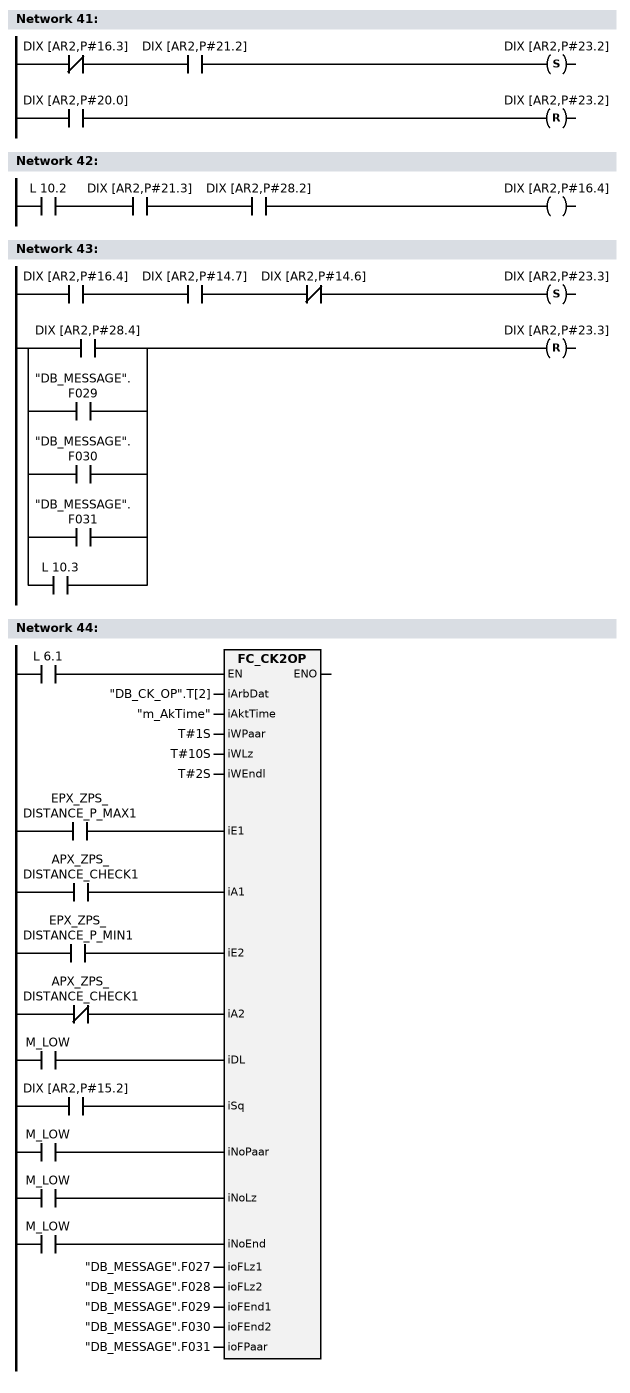
NETWORK
TITLE =
      AN    DIX [AR2,P#16.3];
      A     DIX [AR2,P#21.2];
      S     DIX [AR2,P#23.2];
      A     DIX [AR2,P#20.0];
      R     DIX [AR2,P#23.2];
      NOP   0;
NETWORK
TITLE =
      A     L 10.2;
      A     DIX [AR2,P#21.3];
      A     DIX [AR2,P#28.2];
      =     DIX [AR2,P#16.4];
NETWORK
TITLE =
      A     DIX [AR2,P#16.4];
      A     DIX [AR2,P#14.7];
      AN    DIX [AR2,P#14.6];
      S     DIX [AR2,P#23.3];
      A(;
      O     DIX [AR2,P#28.4];
      O     "DB_MESSAGE".F029;
      O     "DB_MESSAGE".F030;
      O     "DB_MESSAGE".F031;
      O     L 10.3;
      );
      R     DIX [AR2,P#23.3];
      NOP   0;
NETWORK
TITLE =
      A     "EPX_ZPS_DISTANCE_P_MAX1";
      =     L 12.0;
      BLD   103;
      A     "APX_ZPS_DISTANCE_CHECK1";
      =     L 12.1;
      BLD   103;
      A     "EPX_ZPS_DISTANCE_P_MIN1";
      =     L 12.2;
      BLD   103;
      AN    "APX_ZPS_DISTANCE_CHECK1";
      =     L 12.3;
      BLD   103;
      A     "M_LOW";
      =     L 12.4;
      BLD   103;
      A     DIX [AR2,P#15.2];
      =     L 12.5;
      BLD   103;
      A     "M_LOW";
      =     L 12.6;
      BLD   103;
      A     "M_LOW";
      =     L 12.7;
      BLD   103;
      A     "M_LOW";
      =     L 13.0;
      BLD   103;
      A     L 6.1;
      JNB   M014;
      CALL  "FC_CK2OP" (
           iArbDat                  := "DB_CK_OP".T[2],
           iAktTime                 := "m_AkTime",
           iWPaar                   := T#1S,
           iWLz                     := T#10S,
           iWEndl                   := T#2S,
           iE1                      := L 12.0,
           iA1                      := L 12.1,
           iE2                      := L 12.2,
           iA2                      := L 12.3,
           iDL                      := L 12.4,
           iSq                      := L 12.5,
           iNoPaar                  := L 12.6,
           iNoLz                    := L 12.7,
           iNoEnd                   := L 13.0,
           ioFLz1                   := "DB_MESSAGE".F027,
           ioFLz2                   := "DB_MESSAGE".F028,
           ioFEnd1                  := "DB_MESSAGE".F029,
           ioFEnd2                  := "DB_MESSAGE".F030,
           ioFPaar                  := "DB_MESSAGE".F031);
M014: NOP   0;
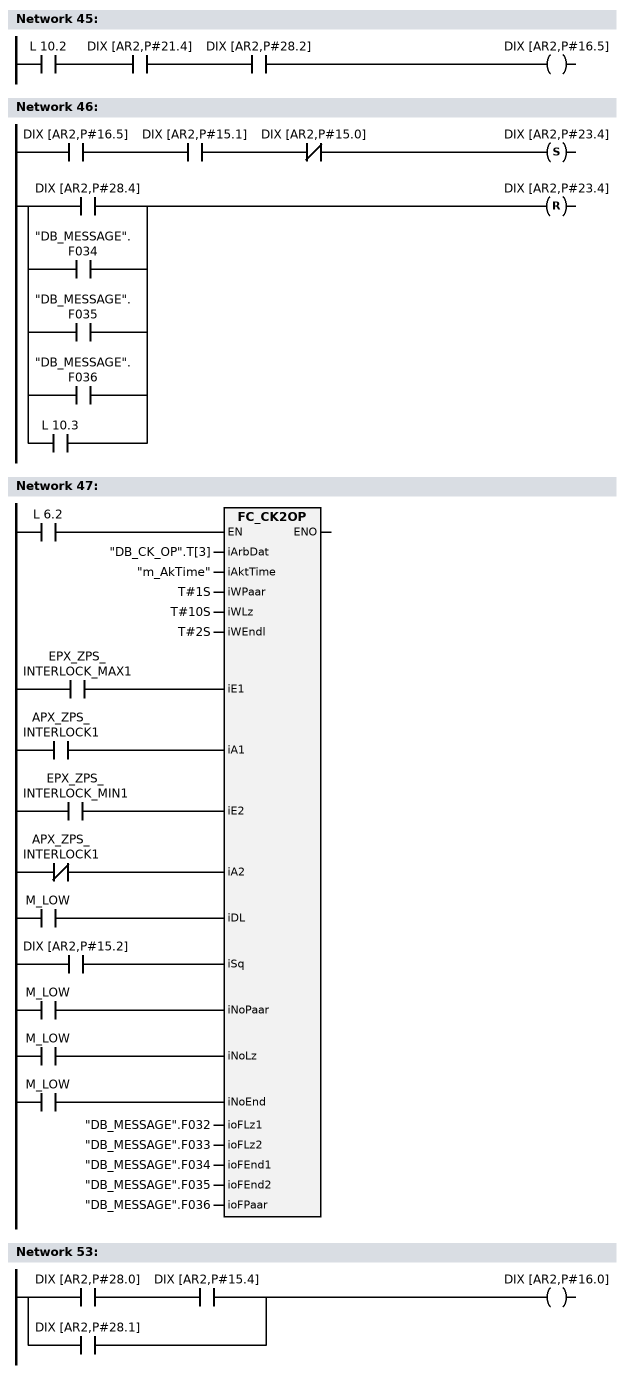
NETWORK
TITLE =
      A     L 10.2;
      A     DIX [AR2,P#21.4];
      A     DIX [AR2,P#28.2];
      =     DIX [AR2,P#16.5];
NETWORK
TITLE =
      A     DIX [AR2,P#16.5];
      A     DIX [AR2,P#15.1];
      AN    DIX [AR2,P#15.0];
      S     DIX [AR2,P#23.4];
      A(;
      O     DIX [AR2,P#28.4];
      O     "DB_MESSAGE".F034;
      O     "DB_MESSAGE".F035;
      O     "DB_MESSAGE".F036;
      O     L 10.3;
      );
      R     DIX [AR2,P#23.4];
      NOP   0;
NETWORK
TITLE =
      A     "EPX_ZPS_INTERLOCK_MAX1";
      =     L 12.0;
      BLD   103;
      A     "APX_ZPS_INTERLOCK1";
      =     L 12.1;
      BLD   103;
      A     "EPX_ZPS_INTERLOCK_MIN1";
      =     L 12.2;
      BLD   103;
      AN    "APX_ZPS_INTERLOCK1";
      =     L 12.3;
      BLD   103;
      A     "M_LOW";
      =     L 12.4;
      BLD   103;
      A     DIX [AR2,P#15.2];
      =     L 12.5;
      BLD   103;
      A     "M_LOW";
      =     L 12.6;
      BLD   103;
      A     "M_LOW";
      =     L 12.7;
      BLD   103;
      A     "M_LOW";
      =     L 13.0;
      BLD   103;
      A     L 6.2;
      JNB   M015;
      CALL  "FC_CK2OP" (
           iArbDat                  := "DB_CK_OP".T[3],
           iAktTime                 := "m_AkTime",
           iWPaar                   := T#1S,
           iWLz                     := T#10S,
           iWEndl                   := T#2S,
           iE1                      := L 12.0,
           iA1                      := L 12.1,
           iE2                      := L 12.2,
           iA2                      := L 12.3,
           iDL                      := L 12.4,
           iSq                      := L 12.5,
           iNoPaar                  := L 12.6,
           iNoLz                    := L 12.7,
           iNoEnd                   := L 13.0,
           ioFLz1                   := "DB_MESSAGE".F032,
           ioFLz2                   := "DB_MESSAGE".F033,
           ioFEnd1                  := "DB_MESSAGE".F034,
           ioFEnd2                  := "DB_MESSAGE".F035,
           ioFPaar                  := "DB_MESSAGE".F036);
M015: NOP   0;
NETWORK
TITLE =
      A     DIX [AR2,P#16.1];
      A     DIX [AR2,P#14.3];
      AN    DIX [AR2,P#14.2];
      A     DIX [AR2,P#16.2];
      A     DIX [AR2,P#14.5];
      AN    DIX [AR2,P#14.4];
      AN    DIX [AR2,P#28.7];
      =     L 10.1;
NETWORK
TITLE =
      A     "M_HIGH";
      =     L 12.0;
      A     L 12.0;
      AN    DIX [AR2,P#28.3];
      AN    DIX [AR2,P#28.5];
      FP    DIX [AR2,P#26.3];
      =     L 11.2;
      A     L 12.0;
      A     L 10.1;
      L     S5T#500MS;
      T     LD 13;
      TAK;
      T     LD 17;
      L     DIW [AR2,P#6.0];
      T     LW 21;
      L     LD 17;
      L     LD 13;
      SD    T [LW 21];
      A     L 12.0;
      A(;
      T     LD 13;
      TAK;
      T     LD 17;
      L     DIW [AR2,P#6.0];
      T     LW 21;
      L     LD 17;
      L     LD 13;
      O     T [LW 21];
      O;
      A     L 10.1;
      T     LD 13;
      TAK;
      T     LD 17;
      L     DIW [AR2,P#8.0];
      T     LW 21;
      L     LD 17;
      L     LD 13;
      A     T [LW 21];
      );
      L     S5T#500MS;
      T     LD 13;
      TAK;
      T     LD 17;
      L     DIW [AR2,P#8.0];
      T     LW 21;
      L     LD 17;
      L     LD 13;
      SF    T [LW 21];
      A     L 11.2;
      T     LD 13;
      TAK;
      T     LD 17;
      L     DIW [AR2,P#8.0];
      T     LW 21;
      L     LD 17;
      L     LD 13;
      R     T [LW 21];
      NOP   0;
      NOP   0;
      T     LD 13;
      TAK;
      T     LD 17;
      L     DIW [AR2,P#8.0];
      T     LW 21;
      L     LD 17;
      L     LD 13;
      A     T [LW 21];
      =     DIX [AR2,P#28.0];
      =     DIX [AR2,P#16.6];
NETWORK
TITLE =
      AN    DIX [AR2,P#16.1];
      AN    DIX [AR2,P#14.3];
      A     DIX [AR2,P#14.2];
      AN    DIX [AR2,P#16.2];
      AN    DIX [AR2,P#14.5];
      A     DIX [AR2,P#14.4];
      AN    DIX [AR2,P#28.6];
      =     L 10.1;
NETWORK
TITLE =
      A     L 10.1;
      A(;
      A(;
      O     DIX [AR2,P#23.3];
      ON    L 6.1;
      );
      A(;
      O     DIX [AR2,P#23.4];
      ON    L 6.2;
      );
      O     DIX [AR2,P#29.0];
      );
      =     L 10.1;
NETWORK
TITLE =
      A     "M_HIGH";
      =     L 12.0;
      A     L 12.0;
      A     L 10.1;
      L     S5T#500MS;
      T     LD 13;
      TAK;
      T     LD 17;
      L     DIW [AR2,P#10.0];
      T     LW 21;
      L     LD 17;
      L     LD 13;
      SD    T [LW 21];
      A     L 12.0;
      A(;
      T     LD 13;
      TAK;
      T     LD 17;
      L     DIW [AR2,P#10.0];
      T     LW 21;
      L     LD 17;
      L     LD 13;
      O     T [LW 21];
      O;
      A     L 10.1;
      T     LD 13;
      TAK;
      T     LD 17;
      L     DIW [AR2,P#12.0];
      T     LW 21;
      L     LD 17;
      L     LD 13;
      A     T [LW 21];
      );
      L     S5T#500MS;
      T     LD 13;
      TAK;
      T     LD 17;
      L     DIW [AR2,P#12.0];
      T     LW 21;
      L     LD 17;
      L     LD 13;
      SF    T [LW 21];
      A     L 11.2;
      T     LD 13;
      TAK;
      T     LD 17;
      L     DIW [AR2,P#12.0];
      T     LW 21;
      L     LD 17;
      L     LD 13;
      R     T [LW 21];
      NOP   0;
      NOP   0;
      T     LD 13;
      TAK;
      T     LD 17;
      L     DIW [AR2,P#12.0];
      T     LW 21;
      L     LD 17;
      L     LD 13;
      A     T [LW 21];
      =     DIX [AR2,P#28.1];
      =     DIX [AR2,P#16.7];
NETWORK
TITLE =
      A     DIX [AR2,P#28.0];
      A     DIX [AR2,P#15.4];
      O     DIX [AR2,P#28.1];
      =     DIX [AR2,P#16.0];
END_FUNCTION_BLOCK

FUNCTION_BLOCK "MESSAGE_OUT"	// FB 100
TITLE = Erfassung Alarm-/Betriebsmeldungen
//________________________________________________________________________________
//$Revision: x.y $
//$Date: 2005/04/26 0:0:0CET $
//$Author: slh $
//$ProjectRevision: Last Checkpoint: m.n $
//
//-------------------------------------------------------------------------------
//*COPYRIGHT BY SCHEUENSTUHL PAC - GERMANY
//*Softwareentwicklung
//erstellt: 27.04.2005; Helmut Scheuenstuhl (slh); Scheuenstuhl PAC
//Änderung: Datum / Abteilung / Name / Version x.y
//Änderung: 
//        :
//Änderung: 19.05.2005 / SPAC / slh / V0.2
//        :a) Neue Funktion:Meldung an die Aufrufebene, wenn ein neuer Eintrag
//        : erfolgt ist (neue E/A's iNEintrAL und oNEintr)
//        :b) Bei neuen Alarm(en) und bisherigen Meldungseinträgen den Stacklese-
//        : zeiger sofort auf den Anfang stellen, um kurzzeitige Alarmnr.-Ausgabe
//        : Wert 0 während laufendem iTimer zu verhindern.
//-------------------------------------------------------------------------------
//Beschreibung
//Der Baustein dient zur Nummerngenerierung von Fehler-/Betriebsmeldungen. Die
//vom Anwenderprg. erzeugten Alarme --- Alarm   001..512   -> DB2.DBX0.0-DBX63.7
//                 bzw. Meldungen ----- Meldung 513..1024  -> DB2.DBX64.0-DBX127.7
//werden mit der fest zugeordneten Nr. erfasst und am Ausgang oAlMldNr wie folgt
//ausgegeben:
//Bei mehreren anstehenden Alarmen/Meldungen werden in einem durch iZeitwert iVm. 
//iTimer festgelegten Zeitraster alle anstehenden Alarme/Meldungen auf oAlMldNr
//durchgeschaltet. Alarme werden höherprior behandelt: Nur wenn kein Alarm 
//ansteht werden Meldungen ausgegeben.
//Eingänge:
//iNEintrAL: Bezieht sich auf oNEintr:Es kann gewählt werden, ob oNEintr nur neue
//         : Alarme melden soll.
//Ausgänge:
//oNEintr : hier wird an die Aufrufebene gemeldet, wenn ein zusätzlicher
//        : Eintrag erfolgt ist (Dauer:1 Plc-Zyklus)
AUTHOR : SPAC_slh
VERSION : 0.2
VAR_INPUT
  IN_TIM_TOGGLE : TIMER ;	//Zeit für Anzeigeintervall
  IN_S5T_TOGGLE : S5TIME ;	//Zeitwert für Anzeigeintervall
  iNEintrAL : BOOL ;	//Ausgabe von oNEintr nur bei Alarmen
END_VAR
VAR_OUTPUT
  OUT_INT_MESSAGENUMBER : INT ;	//Alarm-/Meldungsnr.
  oNEintr : BOOL ;	//Flanke:neuer Eintrag/Alarmeintrag erkannt
  oAlarm : BOOL ;	//Alarm steht an
END_VAR
VAR
  MStack : ARRAY  [0 .. 255 ] OF //Stack für Alarme/Meldungen
  INT ;
  wrStck : INT ;	//Stackzeiger beim Schreiben
  rdStck : INT ;	//Stackzeiger beim Lesen
  wrStckOld : INT ;	//Stackzeigerstand beim Schreiben im letzten Zyklus
  ResInt : INT ;
  ResInt_1 : INT ;
  fk0 : BOOL ;	//Flankenhilfsmerker 0
  x_1 : BOOL ;
  x_2 : BOOL ;
  x_3 : BOOL ;
  x_4 : BOOL ;
  x_5 : BOOL ;
  x_6 : BOOL ;
  x_7 : BOOL ;
  x_8 : BOOL ;
  x_9 : BOOL ;
  x_10 : BOOL ;
  x_11 : BOOL ;
  x_12 : BOOL ;
  x_13 : BOOL ;
  x_14 : BOOL ;
  x_15 : BOOL ;
END_VAR
VAR_TEMP
  svAr1 : DWORD ;	//Rettregister von AR1
  loopctr : INT ;	//Schleifenzähler
  ALMldNr : INT ;	//Alarm-/Meldungsnr.
  PrfWrd : WORD ;	//zu prüfendes Wort
  Bitmaske : WORD ;	//Bitmaske
  Bitnr : BYTE ;	//Bitnr.des gesetzten Bits
  LOp1 : BOOL ;	//lokaler Operationsmerker 1, Zwischenmerker
  fpAlarm : BOOL ;	//pos.Flanke Stack hat einen Alarmeintrag
  StckAlarm : BOOL ;	//Stack hat einen Alarmeintrag
END_VAR
BEGIN
NETWORK
TITLE = Initialisierung, Stack löschen
      OPN   "DB_MESSAGE";
      L     0;
      T     DIW 522;
      TAR1  #svAr1;
      LAR1  P##MStack;
      L     128;
cs01: L     0;
      T     DID [AR1,P#0.0];
      +AR1  P#4.0;
      TAK;
      LOOP  cs01;
NETWORK
TITLE = Erfassung Alarme
      L     0;
s011: T     #loopctr;
      SLW   4;	//slw3:Pointerformat slw1:Wortbreite
      LAR1;
      L     0;
      L     DBW [AR1,P#0.0];
      ==I;
      JC    m011;	//kein Alarmbit gesetzt, nächstes Wort prüfen
      CAW;	//Bytekorrektur
m014: T     #PrfWrd;
      DTR;
      SRD   23;	//im Exponent steht Bias und höchstes gesetztes Bit
      +     -127;	//Bias subtrahieren, bei 32Bit GleitpktZahlen sind das 127
      T     #Bitnr;
      L     #loopctr;
      SLW   4;	//Meldungsoffset pro Wort:hier 16
      +I;
      +     1;	//AlarmnrKorrektur:dbx0.0==Alarmnr.1
//---(1)--- Eintrag in AL-/Meldungspuffer ------------------
      LAR1  P##MStack;
      L     DIW 522;
      SLW   4;	//slw3:Pointerformat slw1:Wortbreite
      +AR1;
      TAK;
      T     DIW [AR1,P#0.0];
      L     255;
      L     DIW 522;
      >I;
      JCN   m013;
      +     1;
      T     DIW 522;
//---(1)----------------------------------------------------
m013: L     0;
      LAR1  P##Bitmaske;
      T     LW [AR1,P#0.0];	//clr Bitmaske
      L     #Bitnr;
      +AR1;
      S     L [AR1,P#0.0];
      L     #Bitmaske;
      CAW;	//Bytekorrektur
      INVI;
      L     #PrfWrd;
      AW;
      L     0;
      <>I;
      TAK;
      JC    m014;	//wenn weiteres Bit gesetzt ist, erneut prüfen
m011: L     31;
      L     #loopctr;
      +     1;
      >=I;
      JC    s011;
NETWORK
TITLE = Erfassung Meldungen
      L     0;
      L     DIW 10;
      <>I;
      =     DIX 8.1;
      =     #StckAlarm;
      JC    m029;	//Wenn schon Eintrag durch Alarme erfolgt, keine Meldungen mehr suchen
      L     32;
s021: T     #loopctr;
      SLW   4;	//slw3:Pointerformat slw1:Wortbreite
      LAR1;
      L     0;
      L     DBW [AR1,P#0.0];
      ==I;
      JC    m021;	//kein Alarmbit gesetzt, nächstes Wort prüfen
      CAW;	//Bytekorrektur
m024: T     #PrfWrd;
      DTR;
      SRD   23;	//im Exponent steht Bias und höchstes gesetztes Bit
      +     -127;	//Bias subtrahieren, bei 32Bit GleitpktZahlen sind das 127
      T     #Bitnr;
      L     #loopctr;
      SLW   4;	//Meldungsoffset pro Wort:hier 16
      +I;
      +     1;	//AlarmnrKorrektur:dbx0.0==Alarmnr.1
//---(1)--- Eintrag in AL-/Meldungspuffer ------------------
      LAR1  P##MStack;
      L     DIW 522;
      SLW   4;	//slw3:Pointerformat slw1:Wortbreite
      +AR1;
      TAK;
      T     DIW [AR1,P#0.0];
      L     255;
      L     DIW 522;
      >I;
      JCN   m023;
      +     1;
      T     DIW 522;
//---(1)----------------------------------------------------
m023: L     0;
      LAR1  P##Bitmaske;
      T     LW [AR1,P#0.0];	//clr Bitmaske
      L     #Bitnr;
      +AR1;
      S     L [AR1,P#0.0];
      L     #Bitmaske;
      CAW;	//Bytekorrektur
      INVI;
      L     #PrfWrd;
      AW;
      L     0;
      <>I;
      TAK;
      JC    m024;	//wenn weiteres Bit gesetzt ist, erneut prüfen
m021: L     63;
      L     #loopctr;
      +     1;
      >=I;
      JC    s021;
m029: NOP   0;
NETWORK
TITLE = pos.Flanke:Stack hat einen Alarmeintrag
      A     #StckAlarm;
      FP    DIX 532.0;
      =     #fpAlarm;
NETWORK
TITLE = Steuerung Stacklesezeiger
      LAR1  #svAr1;
      A(;
      L     0;
      L     DIW 12;
      <>I;
      );
      AN    #fpAlarm;	//wenn bisher MeldAnzeige und ein Alarm neu, sofort rdStck auf Anfang!
      L     DIW 2;
      SD    T [DIW 0];
      JC    m044;
      L     0;
      T     DIW 524;	//rdStck auf Wert 0 setzen wenn keine Meldung ansteht
m044: AN    T [DIW 0];
      JC    m041;
      L     255;
      L     DIW 524;
      +     1;
      <I;
      JCN   m042;
      L     0;
m042: T     DIW 524;
      TAR1  #svAr1;
      LAR1  P##MStack;
      L     DIW 524;
      SLW   4;	//slw3:Pointerformat slw1:Wortbreite
      +AR1;
      L     0;
      L     DIW [AR1,P#0.0];
      ==I;
      LAR1  #svAr1;
      JCN   m043;
      L     0;
      T     DIW 524;	//rdStck auf Wert 0 setzen wenn nächster Platz leer ist
m043: CLR;
      L     DIW 2;
      SD    T [DIW 0];
      SET;
      SD    T [DIW 0];
m041: TAR1  #svAr1;
      LAR1  P##MStack;
      L     DIW 524;
      SLW   4;	//slw3:Pointerformat slw1:Wortbreite
      +AR1;
      L     DIW [AR1,P#0.0];
      LAR1  #svAr1;
      T     #ALMldNr;
NETWORK
TITLE = Ausgang: neuer Eintrag/Alarmeintrag erkannt
      A(;
      A     DIX 4.0;
      A     #StckAlarm;
      ON    DIX 4.0;
      );
      A(;
      L     DIW 526;
      L     DIW 522;
      <I;
      );
      O     #fpAlarm;
      =     DIX 8.0;
      T     DIW 526;
NETWORK
TITLE = Alarm-/Meldungsnr. zur Ausgabe
      L     #ALMldNr;
      T     DIW 6;
END_FUNCTION_BLOCK

FUNCTION "FLOW_CONTROL" : VOID	// FC 10
TITLE = Durchflussüberwachung für KSS im Hoch- oder Niederdruck
//-- IDENTIFIKATION --
// 10 ... Durchflussüberwachung mit Sensor IFM SF5200/VS0200-SN0104
//        --> z.B. Spindel- und Vorschub Halt, wenn Strömung bei aktiver
//            Kühlschmierstofffunktion abreißt.
VERSION : 0.1
VAR_INPUT
  IN_INT_IDENTIFICATION : INT ;	//Auswahl der Funktionalität (...)
  IN_BYT_ANSPRECHZEIT : BYTE ;	//Anwahl der Überwachungszeit beim Einschalten des Mediums
  IN_BYT_ABSCHALTZEIT : BYTE ;	//Anwahl der Überwachungszeit beim Abschalten des Mediums
  IN_BIT_KSS_EIN : BOOL ;	//Kühlschmierstoffzufuhr aktiv
  IN_BIT_DURCHFLUSSWAECHT : BOOL ;	//Schaltsignal des Durchflusswächters
  IN_BIT_LTGUEBERWACHUNG : BOOL ;	//Leitungsüberwachung Durchflusswächter (LOW = Drahtbruch oder Kurzschluß)
  IN_TIM_ANSPRECHZEIT : TIMER ;	//Timer für Ansprechverhalten
  IN_TIM_PRELLEN_ANSPR : TIMER ;	//Timer zum Entprellen des Durchflusswächters
  IN_TIM_ABSCHALTZEIT : TIMER ;	//Timer für Abschaltverhalten
END_VAR
VAR_OUTPUT
  OUT_BIT_DFW_FEHLER : BOOL ;	//Fehler bei Durchflussüberwachung
END_VAR
VAR_IN_OUT
  IO_BIT_FLANKE_1 : BOOL ;	//Hilfsmerker für Flankenauswertung
  I0_BIT_FLANKE_2 : BOOL ;	//Hilfsmerker für Flankenauswertung
  IO_BIT_FLANKE_3 : BOOL ;	//Hilfsmerker für Flankenauswertung
  IO_BIT_HILFSMERKER_KSS : BOOL ;	//Hilfsmerker bei Kühlschmierstoff aus
END_VAR
VAR_TEMP
  TMP_INT_IDENTIFICATION : INT ;	//Identifiaktionsnummer der Funktion
  TMP_INT_ANSPRECHZEIT : INT ;	//Zeitvorwahl - Ansprechzeit
  TMP_INT_ABSCHALTZEIT : INT ;	//Zeitvorwahl - Abschaltzeit
  TMP_S5T_ANSPRECHZEIT : S5TIME ;	//Zeitvariable für Ansprechverhalten
  TMP_S5T_ABSCHALTZEIT : S5TIME ;	//Zeitvariable für Abschaltverhalten
  TMP_BIT_FEHLER_ANSPRECH : BOOL ;	//Fehlerbit - Ansprechverhalten
  TMP_BIT_FEHLER_ABSCHALT : BOOL ;	//Fehlerbit - Abschaltverhalten
  TMP_HILSMERKER_1 : BOOL ;	//Hilfsmerker
  TMP_BIT_ENABLE : BOOL ;	//Bausteinfreigabe - Sammelstörung
END_VAR
BEGIN
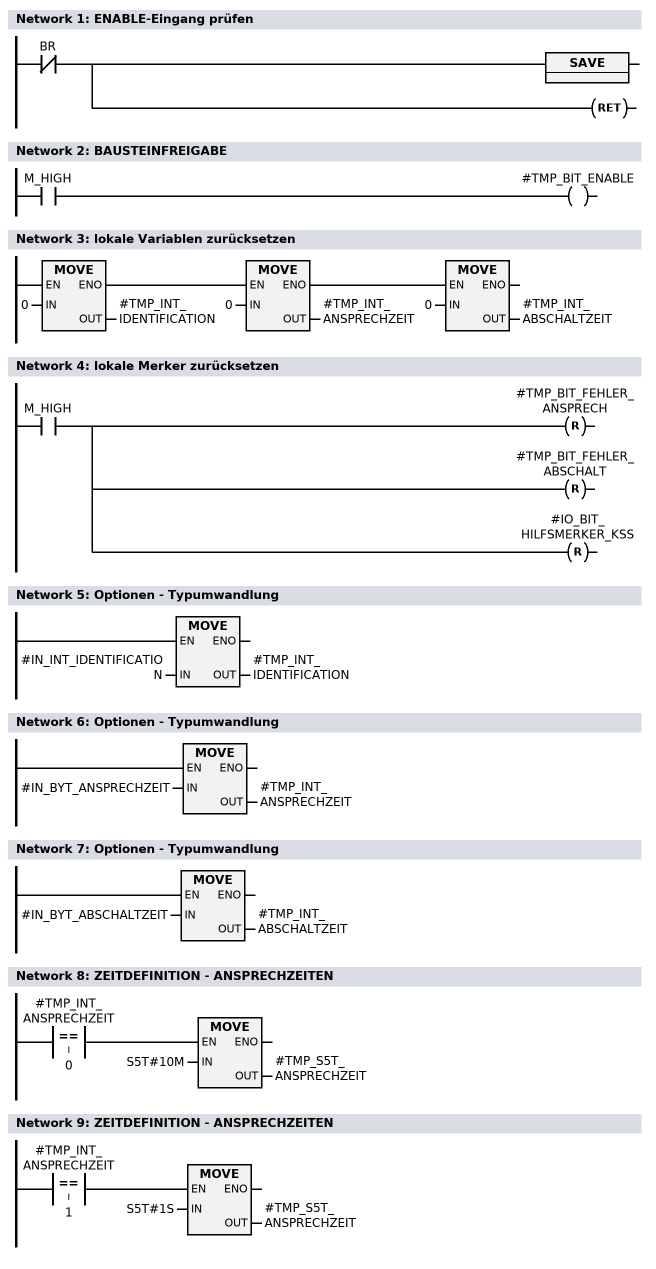
NETWORK
TITLE = ENABLE-Eingang prüfen
//Auswerten des BIE-Statusbit. Dieses entspricht dem EN (ENABLE)-Einganges bei 
//KOP/FUP. Wenn EN=FALSE dann verlasse Baustein.
//
      AN    BR;
      SAVE;
      BEC;
NETWORK
TITLE = BAUSTEINFREIGABE
//Fehlerauswertung Baustein intern:
//Bausteinfreigabe wird gesetzt
      A     "M_HIGH";
      =     #TMP_BIT_ENABLE;
NETWORK
TITLE = lokale Variablen zurücksetzen
      A(;
      A(;
      L     0;
      T     #TMP_INT_IDENTIFICATION;
      SET;
      SAVE;
      CLR;
      A     BR;
      );
      JNB   _001;
      L     0;
      T     #TMP_INT_ANSPRECHZEIT;
      SET;
      SAVE;
      CLR;
_001: A     BR;
      );
      JNB   _002;
      L     0;
      T     #TMP_INT_ABSCHALTZEIT;
_002: NOP   0;
NETWORK
TITLE = lokale Merker zurücksetzen
      A     "M_HIGH";
      R     #TMP_BIT_FEHLER_ANSPRECH;
      R     #TMP_BIT_FEHLER_ABSCHALT;
      R     #IO_BIT_HILFSMERKER_KSS;
NETWORK
TITLE = Optionen - Typumwandlung
//Konvertierung des "Identifikationsbytes" nach Integer
      L     #IN_INT_IDENTIFICATION;
      T     #TMP_INT_IDENTIFICATION;
      NOP   0;
NETWORK
TITLE = Optionen - Typumwandlung
//Konvertierung des "Zeitparameters-Ansprechverhalten" nach Integer
      L     #IN_BYT_ANSPRECHZEIT;
      T     #TMP_INT_ANSPRECHZEIT;
      NOP   0;
NETWORK
TITLE = Optionen - Typumwandlung
//Konvertierung des "Zeitparameters-Abschaltverhalten" nach Integer
      L     #IN_BYT_ABSCHALTZEIT;
      T     #TMP_INT_ABSCHALTZEIT;
      NOP   0;
NETWORK
TITLE = ZEITDEFINITION - ANSPRECHZEITEN
//Zuordnung der Zeit (über Konstante s5T)
//
      A(;
      L     #TMP_INT_ANSPRECHZEIT;
      L     0;
      ==I;
      );
      JNB   _003;
      L     S5T#10M;
      T     #TMP_S5T_ANSPRECHZEIT;
_003: NOP   0;
NETWORK
TITLE = ZEITDEFINITION - ANSPRECHZEITEN
//Zuordnung der Zeit (über Konstante s5T)
      A(;
      L     #TMP_INT_ANSPRECHZEIT;
      L     1;
      ==I;
      );
      JNB   _004;
      L     S5T#1S;
      T     #TMP_S5T_ANSPRECHZEIT;
_004: NOP   0;
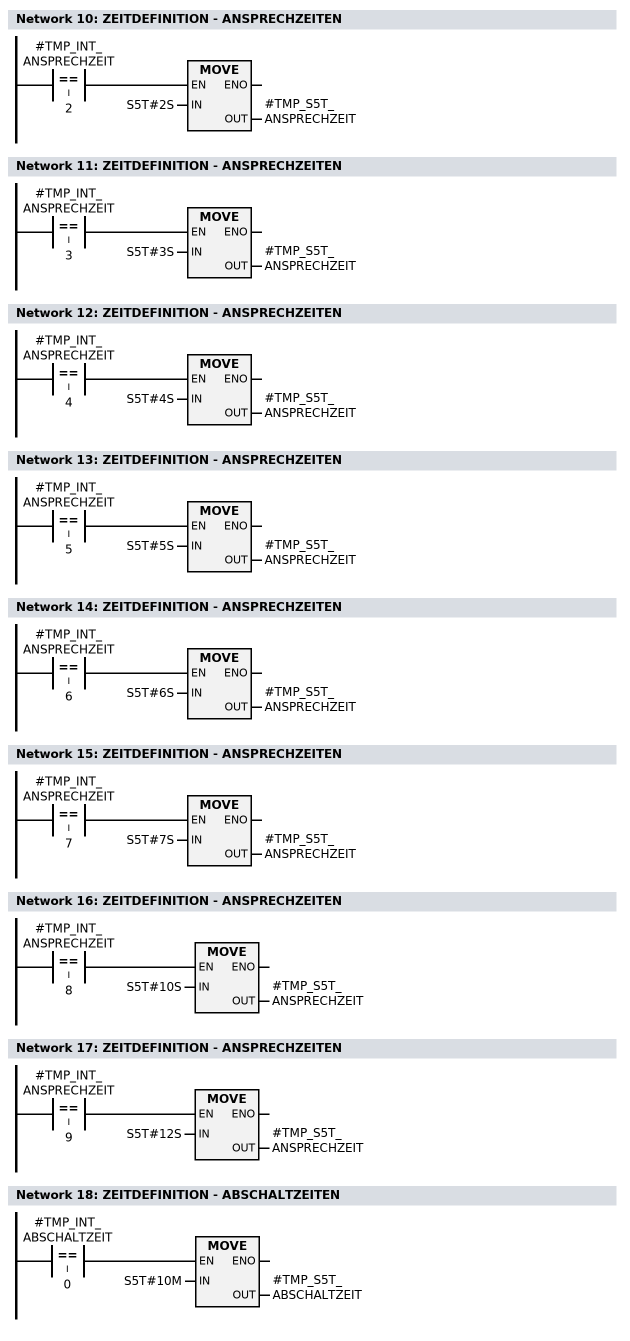
NETWORK
TITLE = ZEITDEFINITION - ANSPRECHZEITEN
//Zuordnung der Zeit (über Konstante s5T)
      A(;
      L     #TMP_INT_ANSPRECHZEIT;
      L     2;
      ==I;
      );
      JNB   _005;
      L     S5T#2S;
      T     #TMP_S5T_ANSPRECHZEIT;
_005: NOP   0;
NETWORK
TITLE = ZEITDEFINITION - ANSPRECHZEITEN
//Zuordnung der Zeit (über Konstante s5T)
      A(;
      L     #TMP_INT_ANSPRECHZEIT;
      L     3;
      ==I;
      );
      JNB   _006;
      L     S5T#3S;
      T     #TMP_S5T_ANSPRECHZEIT;
_006: NOP   0;
NETWORK
TITLE = ZEITDEFINITION - ANSPRECHZEITEN
//Zuordnung der Zeit (über Konstante s5T)
      A(;
      L     #TMP_INT_ANSPRECHZEIT;
      L     4;
      ==I;
      );
      JNB   _007;
      L     S5T#4S;
      T     #TMP_S5T_ANSPRECHZEIT;
_007: NOP   0;
NETWORK
TITLE = ZEITDEFINITION - ANSPRECHZEITEN
//Zuordnung der Zeit (über Konstante s5T)
      A(;
      L     #TMP_INT_ANSPRECHZEIT;
      L     5;
      ==I;
      );
      JNB   _008;
      L     S5T#5S;
      T     #TMP_S5T_ANSPRECHZEIT;
_008: NOP   0;
NETWORK
TITLE = ZEITDEFINITION - ANSPRECHZEITEN
//Zuordnung der Zeit (über Konstante s5T)
      A(;
      L     #TMP_INT_ANSPRECHZEIT;
      L     6;
      ==I;
      );
      JNB   _009;
      L     S5T#6S;
      T     #TMP_S5T_ANSPRECHZEIT;
_009: NOP   0;
NETWORK
TITLE = ZEITDEFINITION - ANSPRECHZEITEN
//Zuordnung der Zeit (über Konstante s5T)
      A(;
      L     #TMP_INT_ANSPRECHZEIT;
      L     7;
      ==I;
      );
      JNB   _00a;
      L     S5T#7S;
      T     #TMP_S5T_ANSPRECHZEIT;
_00a: NOP   0;
NETWORK
TITLE = ZEITDEFINITION - ANSPRECHZEITEN
//Zuordnung der Zeit (über Konstante s5T)
      A(;
      L     #TMP_INT_ANSPRECHZEIT;
      L     8;
      ==I;
      );
      JNB   _00b;
      L     S5T#10S;
      T     #TMP_S5T_ANSPRECHZEIT;
_00b: NOP   0;
NETWORK
TITLE = ZEITDEFINITION - ANSPRECHZEITEN
//Zuordnung der Zeit (über Konstante s5T)
      A(;
      L     #TMP_INT_ANSPRECHZEIT;
      L     9;
      ==I;
      );
      JNB   _00c;
      L     S5T#12S;
      T     #TMP_S5T_ANSPRECHZEIT;
_00c: NOP   0;
NETWORK
TITLE = ZEITDEFINITION - ABSCHALTZEITEN
//Zuordnung der Zeit (über Konstante s5T)
      A(;
      L     #TMP_INT_ABSCHALTZEIT;
      L     0;
      ==I;
      );
      JNB   _00d;
      L     S5T#10M;
      T     #TMP_S5T_ABSCHALTZEIT;
_00d: NOP   0;
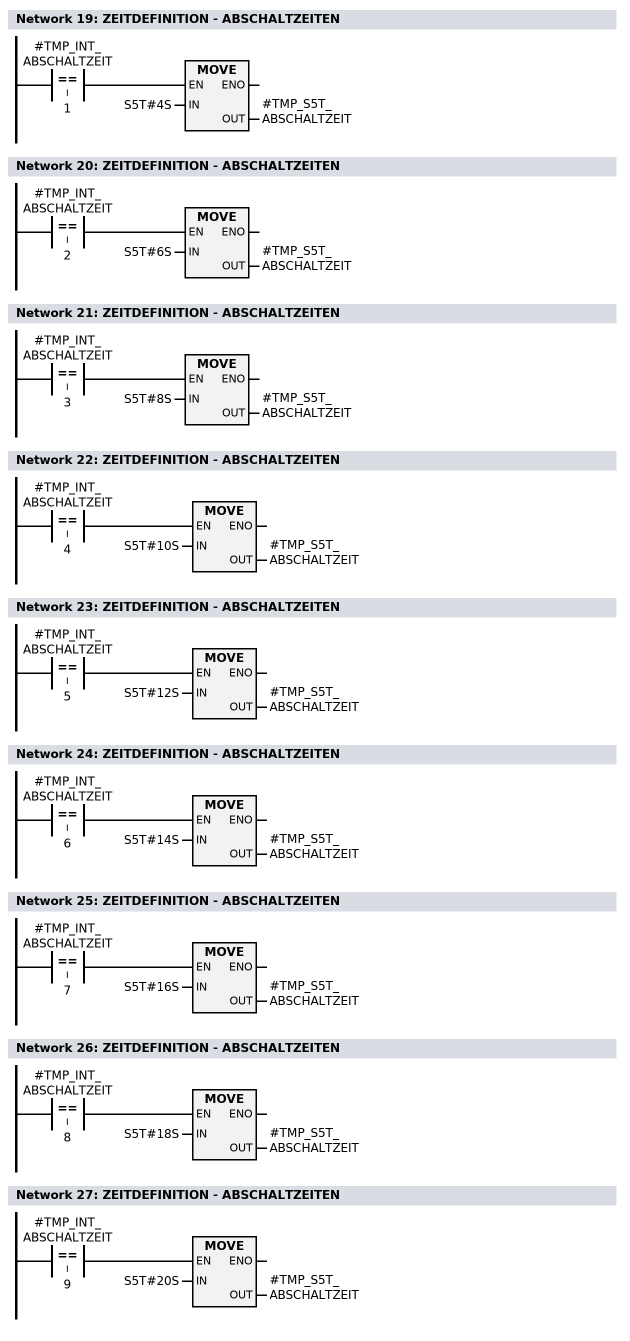
NETWORK
TITLE = ZEITDEFINITION - ABSCHALTZEITEN
//Zuordnung der Zeit (über Konstante s5T)
      A(;
      L     #TMP_INT_ABSCHALTZEIT;
      L     1;
      ==I;
      );
      JNB   _00e;
      L     S5T#4S;
      T     #TMP_S5T_ABSCHALTZEIT;
_00e: NOP   0;
NETWORK
TITLE = ZEITDEFINITION - ABSCHALTZEITEN
//Zuordnung der Zeit (über Konstante s5T)
      A(;
      L     #TMP_INT_ABSCHALTZEIT;
      L     2;
      ==I;
      );
      JNB   _00f;
      L     S5T#6S;
      T     #TMP_S5T_ABSCHALTZEIT;
_00f: NOP   0;
NETWORK
TITLE = ZEITDEFINITION - ABSCHALTZEITEN
//Zuordnung der Zeit (über Konstante s5T)
      A(;
      L     #TMP_INT_ABSCHALTZEIT;
      L     3;
      ==I;
      );
      JNB   _010;
      L     S5T#8S;
      T     #TMP_S5T_ABSCHALTZEIT;
_010: NOP   0;
NETWORK
TITLE = ZEITDEFINITION - ABSCHALTZEITEN
//Zuordnung der Zeit (über Konstante s5T)
      A(;
      L     #TMP_INT_ABSCHALTZEIT;
      L     4;
      ==I;
      );
      JNB   _011;
      L     S5T#10S;
      T     #TMP_S5T_ABSCHALTZEIT;
_011: NOP   0;
NETWORK
TITLE = ZEITDEFINITION - ABSCHALTZEITEN
//Zuordnung der Zeit (über Konstante s5T)
      A(;
      L     #TMP_INT_ABSCHALTZEIT;
      L     5;
      ==I;
      );
      JNB   _012;
      L     S5T#12S;
      T     #TMP_S5T_ABSCHALTZEIT;
_012: NOP   0;
NETWORK
TITLE = ZEITDEFINITION - ABSCHALTZEITEN
//Zuordnung der Zeit (über Konstante s5T)
      A(;
      L     #TMP_INT_ABSCHALTZEIT;
      L     6;
      ==I;
      );
      JNB   _013;
      L     S5T#14S;
      T     #TMP_S5T_ABSCHALTZEIT;
_013: NOP   0;
NETWORK
TITLE = ZEITDEFINITION - ABSCHALTZEITEN
//Zuordnung der Zeit (über Konstante s5T)
      A(;
      L     #TMP_INT_ABSCHALTZEIT;
      L     7;
      ==I;
      );
      JNB   _014;
      L     S5T#16S;
      T     #TMP_S5T_ABSCHALTZEIT;
_014: NOP   0;
NETWORK
TITLE = ZEITDEFINITION - ABSCHALTZEITEN
//Zuordnung der Zeit (über Konstante s5T)
      A(;
      L     #TMP_INT_ABSCHALTZEIT;
      L     8;
      ==I;
      );
      JNB   _015;
      L     S5T#18S;
      T     #TMP_S5T_ABSCHALTZEIT;
_015: NOP   0;
NETWORK
TITLE = ZEITDEFINITION - ABSCHALTZEITEN
//Zuordnung der Zeit (über Konstante s5T)
      A(;
      L     #TMP_INT_ABSCHALTZEIT;
      L     9;
      ==I;
      );
      JNB   _016;
      L     S5T#20S;
      T     #TMP_S5T_ABSCHALTZEIT;
_016: NOP   0;
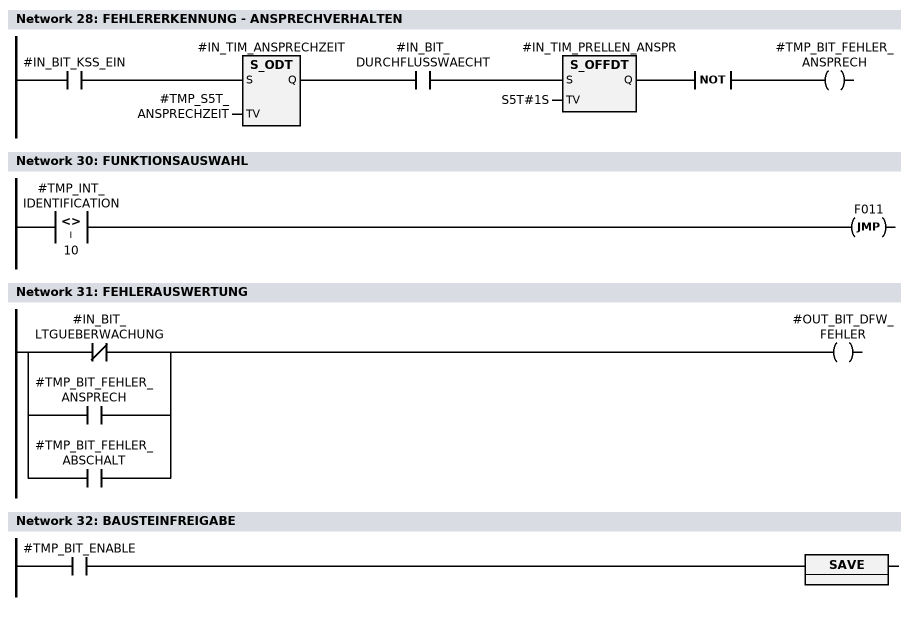
NETWORK
TITLE = FEHLERERKENNUNG - ANSPRECHVERHALTEN
//Das Fehlerbit wird gesetzt, wenn nach Aktivierung der Kühlschmierstoffzufuhr 
//binnen der konfigurierten Zeit <TMP_S5T_ANSPRECHZEIT> der Durchflusswächter 
//nicht durchschaltet. Das Signal des Durchflusswächters wird entprellt 
//<IN_TIM_PRELLEN_ANSPR>. Reißt während der Kühlschmierstoffzufuhr die Strömung 
//ab (Zeit > als Reaktionszeit Sensorik + Entprellzeit), so wird ebenfalls das 
//Fehlerbit gesetzt.
      A(;
      A     #IN_BIT_KSS_EIN;
      L     #TMP_S5T_ANSPRECHZEIT;
      SD    #IN_TIM_ANSPRECHZEIT;
      NOP   0;
      NOP   0;
      NOP   0;
      A     #IN_TIM_ANSPRECHZEIT;
      );
      A(;
      A(;
      A     #IN_BIT_DURCHFLUSSWAECHT;
      L     S5T#1S;
      SF    #IN_TIM_PRELLEN_ANSPR;
      NOP   0;
      NOP   0;
      NOP   0;
      A     #IN_TIM_PRELLEN_ANSPR;
      );
      NOT;
      );
      =     #TMP_BIT_FEHLER_ANSPRECH;
NETWORK
TITLE = FEHLERERKENNUNG - ABSCHALTVERHALTEN
//Das Fehlerbit wird gesetzt, wenn nach Deaktivierung der Kühlschmierstoffzufuhr 
//der Durchflusswächter nicht in der vorgegebenen Zeit <TMP_S5T_ABSCHALTZEIT> 
//zurückschaltet. Über das Flip-Flop (Auswertung der negativen Flanke) wird 
//sichergesetellt, dass die Überwachung nur beim Abschalten des 
//Kühlschmierstoffes wirksam wird.
      A(;
      A     #IN_BIT_KSS_EIN;
      FN    #IO_BIT_FLANKE_1;
      S     #IO_BIT_HILFSMERKER_KSS;
      A(;
      A     #IN_BIT_DURCHFLUSSWAECHT;
      FN    #I0_BIT_FLANKE_2;
      O(;
      A     #IN_BIT_KSS_EIN;
      FP    #IO_BIT_FLANKE_3;
      );
      );
      R     #IO_BIT_HILFSMERKER_KSS;
      A     #IO_BIT_HILFSMERKER_KSS;
      );
      A     #IN_BIT_DURCHFLUSSWAECHT;
      L     #TMP_S5T_ABSCHALTZEIT;
      SD    #IN_TIM_ABSCHALTZEIT;
      NOP   0;
      NOP   0;
      NOP   0;
      A     #IN_TIM_ABSCHALTZEIT;
      =     #TMP_BIT_FEHLER_ABSCHALT;
NETWORK
TITLE = FUNKTIONSAUSWAHL
//Funktionsauswahl für Überwachungsmodus bzw. für Fehlerauswertung
      L     #TMP_INT_IDENTIFICATION;
      L     10;
      <>I;
      JC    F011;
NETWORK
TITLE = FEHLERAUSWERTUNG
//Der Fehlerausgang <OUT_BIT_FEHLER> wird gesetzt, wenn die Leitungsüberwachung
//angesprochen hat oder ein Fehler in der Durchflussüberwachung aufgetreten ist 
//(Ansprech- oder Abschaltverhalten) --> löst z.B. Spindel- und Vorschub Halt aus
      ON    #IN_BIT_LTGUEBERWACHUNG;
      O     #TMP_BIT_FEHLER_ANSPRECH;
      O     #TMP_BIT_FEHLER_ABSCHALT;
      =     #OUT_BIT_DFW_FEHLER;
NETWORK
TITLE = BAUSTEINFREIGABE
//Statusbit BIE=ENO setzen, wenn Funktion ohne Fehler durchlaufen wurde.
F011: A     #TMP_BIT_ENABLE;
      SAVE;
END_FUNCTION

FUNCTION "STATUS_INDICATOR" : VOID	// FC 30
//Konfiguration für spezifische Ausführung von MDE/BDE-Schnittstellen sowie für 
//die Ansteuerung von Signalleuchten.
AUTHOR : A.Petz
VERSION : 0.1
VAR_INPUT
  IN_BYT_IDENTIFICATION : BYTE ;	//Kennung für Funktionsanwahl
END_VAR
VAR_TEMP
  TMP_BIT_ENABLE : BOOL ;	//Bausteinfreigabe - Sammelstörung
  TMP_INT_IDENTIFICATION : INT ;	//Identifiaktionsnummer der Funktion
END_VAR
BEGIN
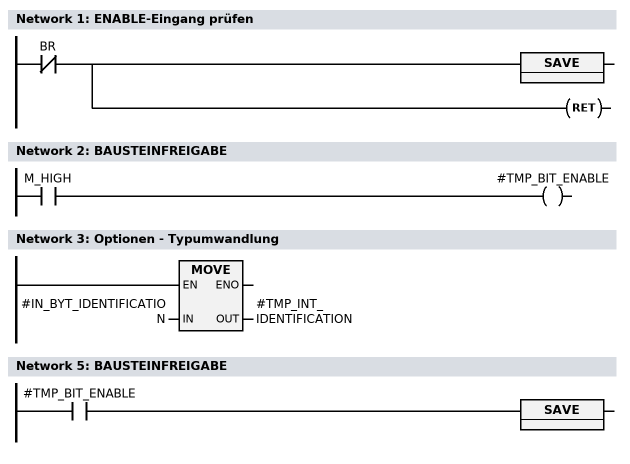
NETWORK
TITLE = ENABLE-Eingang prüfen
//Auswerten des BIE-Statusbit. Dieses entspricht dem EN (ENABLE)-Einganges bei 
//KOP/FUP. Wenn EN=FALSE dann verlasse Baustein.
//
      AN    BR;
      SAVE;
      BEC;
NETWORK
TITLE = BAUSTEINFREIGABE
//Fehlerauswertung Baustein intern:
//Bausteinfreigabe wird gesetzt
      A     "M_HIGH";
      =     #TMP_BIT_ENABLE;
NETWORK
TITLE = Optionen - Typumwandlung
//Konvertierung des "Identifikationsbytes" nach Integer
      L     #IN_BYT_IDENTIFICATION;
      T     #TMP_INT_IDENTIFICATION;
      NOP   0;
NETWORK
TITLE = AUFRUF DER GEWÄHLTEN FUNKTION
//IDENTIFICATION = 10
//Signalleuchte GN/YE/RD
//FC92/2 = Werkzeugmaschine ist in Bearbeitung
//FC92/4 = Fehlermeldung pder Programm Ende
      L     #TMP_INT_IDENTIFICATION;
      L     10;
      ==I;
      =     L 4.0;
      A     L 4.0;
      JNB   _001;
      CALL  "SIGNAL" (
           IN_INT_IDENTIFICATION    := 2,
           OUT_BIT_SIGNAL           := "APX_SIGNAL_TOWER_GN");	//"SIGNAL"
_001: NOP   0;
      A     L 4.0;
      AN    "APX_SIGNAL_TOWER_GN";
      O     DB111.DBX 6.0;
      O;
      A     DB111.DBX 6.1;
      A     "M_TAKT_0.5SEC";
      =     "APX_SIGNAL_TOWER_YE";
      A     L 4.0;
      JNB   _002;
      CALL  "SIGNAL" (
           IN_INT_IDENTIFICATION    := 4,
           OUT_BIT_SIGNAL           := "APX_SIGNAL_TOWER_RD");
_002: NOP   0;
NETWORK
TITLE = BAUSTEINFREIGABE
//Statusbit BIE=ENO setzen, wenn Funktion ohne Fehler durchlaufen wurde.
      A     #TMP_BIT_ENABLE;
      SAVE;
END_FUNCTION

